// TwinCAT 3 PLC project UnitTests
// ProgramVersion: 3.1.4026.27
// libraries:
//   [ApplicationBase], * (Beckhoff Automation LLC)
//   Tc2_EtherCAT, * (Beckhoff Automation GmbH)
//   Tc2_Math, * (Beckhoff Automation GmbH)
//   Tc2_MC2, * (Beckhoff Automation GmbH)
//   Tc2_Standard, * (Beckhoff Automation GmbH)
//   Tc2_System, * (Beckhoff Automation GmbH)
//   Tc2_Utilities, * (Beckhoff Automation GmbH)
//   Tc3_EventLogger, * (Beckhoff Automation GmbH)
//   Tc3_PlcTestSuite, * (Simmel)
// project tree:
//   / TestsBase.TcPOU, TestsBaseTask.TcTTO
//   UnitTests/ADS/ ADS_TEST.TcPOU
//   UnitTests/Analog/ Analog_TEST.TcPOU
//   UnitTests/AnyBuffer/ AnyBuffer_TEST.TcPOU, GVL_TEST_AnyBuffer.TcGVL, TEST_AnyBuffer_Clear.TcPOU, TEST_AnyBuffer_DeleteAtIndex.TcPOU, TEST_AnyBuffer_InsertAtIndex.TcPOU, TEST_AnyBuffer_PeekAtIndex.TcPOU, TEST_AnyBuffer_PopAtIndex.TcPOU, TEST_AnyBuffer_PopLeft.TcPOU, TEST_AnyBuffer_PopRight.TcPOU, TEST_AnyBuffer_PushLeft.TcPOU, TEST_AnyBuffer_PushRight.TcPOU, TEST_AnyBuffer_ReplaceAtIndex.TcPOU
//   UnitTests/AnyBuffer/DUTs/ ST_TEST_AnyBuffer_Element.TcDUT
//   UnitTests/Axis/ Axis_Test.TcPOU
//   UnitTests/CollectionPeeker/ CollectionPeeker_Test.TcPOU
//   UnitTests/Collection/ Collection_TEST.TcPOU
//   UnitTests/ComponentCollection/ ComponentCollection_TEST.TcPOU
//   UnitTests/Component/ Component_TEST.TcPOU
//   UnitTests/CyclicComponent/ CyclicComponent_TEST.TcPOU
//   UnitTests/CyclicRunner/ CyclicRunner_TEST.TcPOU
//   UnitTests/Cylinder/ Cylinder_TEST.TcPOU
//   UnitTests/Digital/ DigitalInput_Combiner_TEST.TcPOU, DigitalInput_Debounce_TEST.TcPOU, DigitalInput_ForceVisitor_TEST.TcPOU, DigitalInput_NC_TEST.TcPOU, DigitalInput_NO_TEST.TcPOU, DigitalOutput_TEST.TcPOU
//   UnitTests/Events/ Events_TEST.TcPOU
//   UnitTests/EtherCat/ EtherCatMaster_TEST.TcPOU
//   UnitTests/Force/ ForcibleBool_TEST.TcPOU, ForcibleInt_Test.TcPOU
//   UnitTests/Initializer/ Initializer_TEST.TcPOU
//   UnitTests/List/ List_TEST.TcPOU
//   UnitTests/ModeChange/ ModeControl_TEST.TcPOU
//   UnitTests/ModuleCollection/ ModuleCollection_TEST.TcPOU
//   UnitTests/Module/ Module_TEST.TcPOU
//   UnitTests/Recipe/ Recipe_TEST.TcPOU, ST_Recipe.TcDUT
//   UnitTests/Safety/ SafetyBase_TEST.TcPOU
//   UnitTests/Serial/ SerialConnection_Tests.TcPOU
//   UnitTests/Statemachine/ Statemachine_TEST.TcPOU
//   UnitTests/Tracing/ Tracing_TEST.TcPOU
//   UnitTests/Utilities/ Utilities_TEST.TcPOU
//   _Mockups/AnyBuffer/ GVL_Samples_AnyBuffer.TcGVL, SampleFifo.TcPOU, SampleLifo.TcPOU, SampleList.TcPOU, SampleRing.TcPOU, Samples_AnyBuffer.TcPOU
//   _Mockups/CollectionPeeker/ CollectionPeeker_Mock.TcPOU
//   _Mockups/Collection/ Collection_Mockup.TcPOU, Item_Mockup.TcPOU
//   _Mockups/Components/ Component_Mockup.TcPOU, CyclicComponent_Mockup.TcPOU, InitializableComponent_Mockup.TcPOU, MockupComponentTcEvent.TcPOU
//   _Mockups/EtherCat/ EtherCatEventProvider_Mockup.TcPOU, EtherCatMaster_Mockup.TcPOU
//   _Mockups/ModeChange/ ModeControl_Mockup.TcPOU
//   _Mockups/Modules/ EquipmentModule_Mockup.TcPOU, MachineModule_Mockup.TcPOU, ModuleCollection_Mockup.TcPOU, Module_Mockup.TcPOU
//   _Mockups/SerialLineCtrl/ MockSerialLineCtrl.TcPOU
//   _Mockups/Statemachine/ StateMachineVisitor_Mockup.TcPOU, State_Mockup.TcPOU
//   _Mockups/Visitors/ ComponentVisitor_Mockup.TcPOU, GetSystemTreeNamesVisitor.TcPOU, ModuleVisitor_Mockup.TcPOU, QueryInterfaceResettables.TcPOU, StringCollection.TcPOU
// real-time tasks:
//   TASK UnitTestsBase: cycle T#10ms, priority 20, ADS port 350
//   TASK VFFS: cycle T#10ms, priority 21, ADS port 351
//   TASK PlcTask: cycle T#10ms, priority 22, ADS port 352
//   TASK Job Task: cycle default, priority 32
//   TASK MC-Task (MET): cycle T#2ms, priority 3, ADS port 521
//   TASK MC-Task (MPT): cycle T#10ms, priority 9, ADS port 531
// motion (NC):
//   TASK NC-Task 1 SAF: cycle T#2ms, priority 4, ADS port 501
//   TASK NC-Task 1 SVB: cycle T#10ms, priority 8, ADS port 511
//   AXIS TestAxis (id 1)
//     OtherSettings: AllowMotionCmdToSlave=true
//     encoder EncType=1
//     drive DrvType=5
//       Analog: TorqueSetpointScale=10, ScaleFactorActTorque=0.1
//     controller CtrType=1
//       CtrPara: PriorControlFactor=1
//         Observer: BandWidth=20
//   AXIS Unwind (id 2)
//     OtherSettings: AllowMotionCmdToSlave=true
//     encoder EncType=1
//     drive DrvType=5
//       Analog: TorqueSetpointScale=10, ScaleFactorActTorque=0.1
//       TimeComp: TaskDelayCycles=1
//     controller CtrType=1
//       CtrPara: PriorControlFactor=1
//         Observer: BandWidth=20
//   AXIS Seal (id 3)
//     OtherSettings: AllowMotionCmdToSlave=true
//     encoder EncType=1
//     drive DrvType=5
//       Analog: TorqueSetpointScale=10, ScaleFactorActTorque=0.1
//       TimeComp: TaskDelayCycles=1
//     controller CtrType=1
//       CtrPara: PriorControlFactor=1
//         Observer: BandWidth=20
//   AXIS Pull Wheel Left (id 4)
//     OtherSettings: AllowMotionCmdToSlave=true
//     encoder EncType=1
//     drive DrvType=5
//       Analog: TorqueSetpointScale=10, ScaleFactorActTorque=0.1
//       TimeComp: TaskDelayCycles=1
//     controller CtrType=1
//       CtrPara: PriorControlFactor=1
//         Observer: BandWidth=20
//   AXIS Pull Wheel Right (id 5)
//     OtherSettings: AllowMotionCmdToSlave=true
//     encoder EncType=1
//     drive DrvType=5
//       Analog: TorqueSetpointScale=10, ScaleFactorActTorque=0.1
//       TimeComp: TaskDelayCycles=1
//     controller CtrType=1
//       CtrPara: PriorControlFactor=1
//         Observer: BandWidth=20
// variable links:
//   (this object) <-> NC-Task 1 SAF/Axes/TestAxis
//     TestsBaseTask Inputs/TestsBase.Axis_Test.AxisRef.NcToPlc <-> Outputs/ToPlc
//     TestsBaseTask Outputs/TestsBase.Axis_Test.AxisRef.PlcToNc <-> Inputs/FromPlc
//   (this object) <-> UnitTests/UnitTests Instance
//     TestsBaseTask Inputs/TestsBase.SafetyBase_TEST.EStop_NOK.InfoData/Diag <-> TestsBaseTask Outputs/TestsBase.SafetyBase_TEST.InfoData_NOK/Diag
//     TestsBaseTask Inputs/TestsBase.SafetyBase_TEST.EStop_NOK.InfoData/State <-> TestsBaseTask Outputs/TestsBase.SafetyBase_TEST.InfoData_NOK/State
//     TestsBaseTask Inputs/TestsBase.SafetyBase_TEST.EStop_OK.InfoData/Diag <-> TestsBaseTask Outputs/TestsBase.SafetyBase_TEST.InfoData_OK/Diag
//     TestsBaseTask Inputs/TestsBase.SafetyBase_TEST.EStop_OK.InfoData/State <-> TestsBaseTask Outputs/TestsBase.SafetyBase_TEST.InfoData_OK/State
//     TestsBaseTask Inputs/TestsBase.SafetyBase_TEST.EStop_Sim.InfoData/Diag <-> TestsBaseTask Outputs/TestsBase.SafetyBase_TEST.InfoData_OK/Diag
//     TestsBaseTask Inputs/TestsBase.SafetyBase_TEST.EStop_Sim.InfoData/State <-> TestsBaseTask Outputs/TestsBase.SafetyBase_TEST.InfoData_OK/State
//     TestsBaseTask Inputs/TestsBase.SafetyBase_TEST.Group.InfoData/Diag <-> TestsBaseTask Outputs/TestsBase.SafetyBase_TEST.InfoData_Group/Diag
//     TestsBaseTask Inputs/TestsBase.SafetyBase_TEST.Group.InfoData/State <-> TestsBaseTask Outputs/TestsBase.SafetyBase_TEST.InfoData_Group/State
//     TestsBaseTask Inputs/TestsBase.SafetyBase_TEST.Reset <-> TestsBaseTask Outputs/TestsBase.SafetyBase_TEST.ResetPulse.Reset
//     TestsBaseTask Inputs/TestsBase.SafetyBase_TEST.Run <-> TestsBaseTask Outputs/TestsBase.SafetyBase_TEST.Group.Run
//     TestsBaseTask Outputs/TestsBase.SafetyBase_TEST.Group.Run <-> TestsBaseTask Inputs/TestsBase.SafetyBase_TEST.Run
//     TestsBaseTask Outputs/TestsBase.SafetyBase_TEST.InfoData_Group/Diag <-> TestsBaseTask Inputs/TestsBase.SafetyBase_TEST.Group.InfoData/Diag
//     TestsBaseTask Outputs/TestsBase.SafetyBase_TEST.InfoData_Group/State <-> TestsBaseTask Inputs/TestsBase.SafetyBase_TEST.Group.InfoData/State
//     TestsBaseTask Outputs/TestsBase.SafetyBase_TEST.InfoData_NOK/Diag <-> TestsBaseTask Inputs/TestsBase.SafetyBase_TEST.EStop_NOK.InfoData/Diag
//     TestsBaseTask Outputs/TestsBase.SafetyBase_TEST.InfoData_NOK/State <-> TestsBaseTask Inputs/TestsBase.SafetyBase_TEST.EStop_NOK.InfoData/State
//     TestsBaseTask Outputs/TestsBase.SafetyBase_TEST.InfoData_OK/Diag <-> TestsBaseTask Inputs/TestsBase.SafetyBase_TEST.EStop_OK.InfoData/Diag
//     TestsBaseTask Outputs/TestsBase.SafetyBase_TEST.InfoData_OK/Diag <-> TestsBaseTask Inputs/TestsBase.SafetyBase_TEST.EStop_Sim.InfoData/Diag
//     TestsBaseTask Outputs/TestsBase.SafetyBase_TEST.InfoData_OK/State <-> TestsBaseTask Inputs/TestsBase.SafetyBase_TEST.EStop_OK.InfoData/State
//     TestsBaseTask Outputs/TestsBase.SafetyBase_TEST.InfoData_OK/State <-> TestsBaseTask Inputs/TestsBase.SafetyBase_TEST.EStop_Sim.InfoData/State
//     TestsBaseTask Outputs/TestsBase.SafetyBase_TEST.ResetPulse.Reset <-> TestsBaseTask Inputs/TestsBase.SafetyBase_TEST.Reset
//   (this object) <-> MC Project1/Axes/Pull Wheel Left
//     PlcTask Inputs/MAIN.VFFS._PullWheels.PullWheelLeftAxisRef.McToPlc/Act <-> McToPlc/Act
//     PlcTask Inputs/MAIN.VFFS._PullWheels.PullWheelLeftAxisRef.McToPlc/Set <-> McToPlc/Set
//     PlcTask Inputs/MAIN.VFFS._PullWheels.PullWheelLeftAxisRef.McToPlc/Std <-> McToPlc/Std
//     PlcTask Outputs/MAIN.VFFS._PullWheels.PullWheelLeftAxisRef.PlcToMc/Std <-> PlcToMc/Std
//   (this object) <-> MC Project1/Axes/Pull Wheel Right
//     PlcTask Inputs/MAIN.VFFS._PullWheels.PullWheelRightAxisRef.McToPlc/Act <-> McToPlc/Act
//     PlcTask Inputs/MAIN.VFFS._PullWheels.PullWheelRightAxisRef.McToPlc/Set <-> McToPlc/Set
//     PlcTask Inputs/MAIN.VFFS._PullWheels.PullWheelRightAxisRef.McToPlc/Std <-> McToPlc/Std
//     PlcTask Outputs/MAIN.VFFS._PullWheels.PullWheelRightAxisRef.PlcToMc/Std <-> PlcToMc/Std
//   (this object) <-> MC Project1/Axes/Seal
//     PlcTask Inputs/MAIN.VFFS._Sealer.SealerAxisRef.McToPlc/Act <-> McToPlc/Act
//     PlcTask Inputs/MAIN.VFFS._Sealer.SealerAxisRef.McToPlc/Set <-> McToPlc/Set
//     PlcTask Inputs/MAIN.VFFS._Sealer.SealerAxisRef.McToPlc/Std <-> McToPlc/Std
//     PlcTask Outputs/MAIN.VFFS._Sealer.SealerAxisRef.PlcToMc/Std <-> PlcToMc/Std
//   (this object) <-> MC Project1/Axes/Unwind
//     PlcTask Inputs/MAIN.VFFS._Unwind.UnwindAxisRef.McToPlc/Act <-> McToPlc/Act
//     PlcTask Inputs/MAIN.VFFS._Unwind.UnwindAxisRef.McToPlc/Set <-> McToPlc/Set
//     PlcTask Inputs/MAIN.VFFS._Unwind.UnwindAxisRef.McToPlc/Std <-> McToPlc/Std
//     PlcTask Outputs/MAIN.VFFS._Unwind.UnwindAxisRef.PlcToMc/Std <-> PlcToMc/Std

CONFIGURATION UnitTests
    RESOURCE PLC ON TwinCAT3
        TASK TestsBaseTask(INTERVAL := T#10ms, PRIORITY := 20);
        PROGRAM TestsBase WITH TestsBaseTask : TestsBase;
    END_RESOURCE
END_CONFIGURATION

// ---- UnitTests/AnyBuffer/DUTs/ST_TEST_AnyBuffer_Element.TcDUT
TYPE ST_TEST_AnyBuffer_Element :
STRUCT
	id				: INT;
	name			: STRING;
END_STRUCT
END_TYPE

// ---- UnitTests/Recipe/ST_Recipe.TcDUT
TYPE ST_Recipe :
	STRUCT
		ValueA : LREAL;
		ValueB : DINT;
		ValueC : BOOL;
	END_STRUCT
END_TYPE

// ---- UnitTests/AnyBuffer/GVL_TEST_AnyBuffer.TcGVL
VAR_GLOBAL
	// System Under Test (SUT)
    RawBuffer       		: ARRAY[TEST_LL..TEST_UL] OF DINT;
    fbAnyBuffer    			: AnyBuffer(pBuffer := RawBuffer,
									bufferBoundLower := TEST_LL,
									bufferBoundUpper := TEST_UL,
									isBufferPersistent := FALSE);

	// Compare buffer
	CompareBuffer : ARRAY[TEST_LL..TEST_UL] OF DINT;
	fbCompareBuffer : AnyBuffer(pBuffer := CompareBuffer,
								bufferBoundLower := TEST_LL,
								bufferBoundUpper := TEST_UL,
								isBufferPersistent := FALSE);

    // Test Variables
    Success         		: BOOL;
	AppendedElement			: DINT;
	ReturnedElement			: DINT;
	WrongSizeElement		: INT;
	testElement				: DINT;

	// Bool
	TEST_BOOL_TRUE			: BOOL := TRUE;
	TEST_BOOL_FALSE			: BOOL := FALSE;
	TEST_DINT				: DINT;
	TEST_REAL				: REAL;
END_VAR
VAR_GLOBAL CONSTANT
	// Changing the limits is allowed, but the tests are built for an array size 5 elements
	TEST_LL					: INT := 0;
	TEST_UL					: INT := 4;
END_VAR

// ---- _Mockups/AnyBuffer/GVL_Samples_AnyBuffer.TcGVL
VAR_GLOBAL PERSISTENT
	buffer					: ARRAY[S_LL..S_UL] OF ST_TEST_AnyBuffer_Element;			// Any size buffer of any type
END_VAR

VAR_GLOBAL
	anyBuffer				: AnyBuffer(buffer, S_LL, S_UL, TRUE); 		// persistent buffer handler
END_VAR

VAR_GLOBAL CONSTANT
	S_LL					: INT := 0;
	S_UL					: INT := 2;
END_VAR

// ---- TestsBase.TcPOU
PROGRAM TestsBase
VAR
	CyclicRunner_TEST			   : CyclicRunner_TEST;
	ComponentCollection_TEST	   : ComponentCollection_TEST;
	Module_TEST					   : Module_TEST;
	CyclicComponent_TEST		   : CyclicComponent_TEST;
	Component_TEST				   : Component_TEST;
	ModuleCollection_TEST		   : ModuleCollection_TEST;
	Tracing_TEST				   : Tracing_TEST;
	Initializer_TEST			   : Initializer_TEST;
	Events_TEST					   : Events_TEST;
	Statemachine_TEST			   : Statemachine_TEST;
	Collection_Test				   : Collection_TEST();
	List_TEST					   : List_TEST;
	ModeControl_TEST			   : ModeControl_TEST;
	CollectionPeeker_Test		   : CollectionPeeker_Test;
	ForcibleBool_TEST			   : ForcibleBool_TEST;
	ForcibleInt_Test			   : ForcibleInt_Test;
	Utilities_TEST				   : Utilities_TEST;
	DigitalInput_NC_TEST		   : DigitalInput_NC_TEST;
	DigitalInput_NO_TEST		   : DigitalInput_NO_TEST;
	DigitalOutput_TEST			   : DigitalOutput_TEST;
	DigitalInput_Combiner_TEST	   : DigitalInput_Combiner_TEST;
	DigitalInput_Debounce_TEST	   : DigitalInput_Debounce_TEST;
	Cylinder_TEST				   : Cylinder_TEST;
	SafetyBase_TEST				   : SafetyBase_TEST;
	ADS_TEST					   : ADS_TEST;
	DigitalInput_ForceVisitor_TEST : DigitalInput_ForceVisitor_TEST;
	Recipe_TEST					   : Recipe_TEST;
	Analog_TEST					   : Analog_TEST;
	Serial_TEST					   : SerialConnection_Tests;
	Axis_Test					   : Axis_Test;
	EtherCatMaster_TEST		   : EtherCatMaster_TEST;

	//
	Component1				  : CyclicComponent_Mockup('Component 1');
	Component2				  : CyclicComponent_Mockup('Component 2');
	Component3				  : CyclicComponent_Mockup('Component 3');
	Component4				  : CyclicComponent_Mockup('Component 4');
	Em						  : EquipmentModule_Mockup('Em', Component1, Component2);
	EmEm					  : MachineModule_Mockup('EmEm', Em, Component3, Component4);
	EmEmEm					  : MachineModule_Mockup('EmEmEm', EmEm, Component3, Component4);
	Machine					  : MachineModule_Mockup('Machine', EmEmEm, Component3, Component4);
	StringCollection		  : StringCollection<100>;
	MachineModuleVisitor	  : GetSystemTreeNamesVisitor(StringCollection);
	QueryInterfaceResettables : QueryInterfaceResettables();
	Rerun					  : BOOL;
END_VAR

GlobalTestSuite.TestSuite.TestSuiteName := 'Application Base Test Suite';
Tracing_TEST();
CyclicRunner_TEST();
ComponentCollection_TEST();
Module_TEST();
Component_TEST();
CyclicComponent_TEST();
ModuleCollection_TEST();
Initializer_TEST();
Events_TEST();
Statemachine_TEST();
Collection_Test();
List_TEST();
ModeControl_TEST();
CollectionPeeker_Test();
ForcibleBool_TEST();
Utilities_TEST();
DigitalInput_NC_TEST();
DigitalInput_NO_TEST();
DigitalOutput_TEST();
DigitalInput_Combiner_TEST();
DigitalInput_Debounce_TEST();
Cylinder_TEST();
SafetyBase_TEST();
ADS_TEST();
DigitalInput_ForceVisitor_TEST();
Recipe_TEST();
Analog_TEST();
AnyBuffer_TEST();
ForcibleInt_Test();
Serial_TEST();
Axis_Test();
EtherCatMaster_TEST();

// Mockup code
Samples_AnyBuffer();
//
IF NOT Machine.Initialized THEN
	Machine.Initialize();
ELSE
	Machine.CyclicLogic();
	MachineModuleVisitor.GetTree(Machine);
	QueryInterfaceResettables.GetAllResetComponents(Em);
END_IF

IF Rerun THEN
	Rerun := FALSE;
	GlobalTestSuite.TestSuite.ReRunTests();
END_IF

END_PROGRAM

// ---- UnitTests/CyclicRunner/CyclicRunner_TEST.TcPOU
FUNCTION_BLOCK CyclicRunner_TEST
VAR
END_VAR

AddTwoCyclicCalleesAndRun();
CollectionAddsCyclicSucessfully();
CollectionRejectsAddingCyclicDuplicate();
CollectionRejectsAddingNullCyclic();
CollectionRejectsAddingTooManyCyclics();
CollectionRejectsRemoveWhenEmpty();
CollectionRejectsRemoveWhenNotFound();
CollectionRejectsRemovingNullCyclic();
CollectionRemovesCyclicSuccessfully();

METHOD AddTwoCyclicCalleesAndRun
VAR
	Expected	 : BOOL := TRUE;
	Actual		 : BOOL;
	CyclicRunner : CyclicRunner<ApplicationBaseParameter.MaxCountInCollections>;
	Component	 : ARRAY[0..1] OF CyclicComponent_Mockup[(Name := 'Component 1'), (Name := 'Component 2')];
END_VAR
IF TestSuite.Test(__POUNAME()).ExecuteTest() THEN
	CyclicRunner.AddCallee(Component[0]);
	CyclicRunner.AddCallee(Component[1]);
	CyclicRunner.CallAll();
	Actual := Component[0].WasCalled AND Component[1].WasCalled;
	TestSuite.Test(__POUNAME()).AssertEqual(Expected, Actual);
END_IF
END_METHOD

METHOD CollectionAddsCyclicSucessfully
VAR
	Expected	   : BOOL := TRUE;
	Actual		   : BOOL;
	CyclicRunner : CyclicRunner<ApplicationBaseParameter.MaxCountInCollections>;
	Cyclic	 : CyclicComponent_Mockup(Name := 'Cyclic 1');
END_VAR
IF TestSuite.Test(__POUNAME()).ExecuteTest() THEN
	Actual := CyclicRunner.AddCallee(Cyclic) = RegistrationResult.Succeeded;
	TestSuite.Test(__POUNAME()).AssertEqual(Expected, Actual);
END_IF
END_METHOD

METHOD CollectionRejectsAddingCyclicDuplicate
VAR
	Expected	   : BOOL := TRUE;
	Actual		   : BOOL;
	CyclicRunner : CyclicRunner<ApplicationBaseParameter.MaxCountInCollections>;
	Cyclic	 : CyclicComponent_Mockup(Name := 'Cyclic 1');
END_VAR
IF TestSuite.Test(__POUNAME()).ExecuteTest() THEN
	CyclicRunner.AddCallee(Cyclic);
	Actual := CyclicRunner.AddCallee(Cyclic) = RegistrationResult.AlreadyAdded;
	TestSuite.Test(__POUNAME()).AssertEqual(Expected, Actual);
END_IF
END_METHOD

METHOD CollectionRejectsAddingNullCyclic
VAR
	Expected	   : BOOL := TRUE;
	Actual		   : BOOL;
	CyclicRunner : CyclicRunner<ApplicationBaseParameter.MaxCountInCollections>;
END_VAR
IF TestSuite.Test(__POUNAME()).ExecuteTest() THEN
	Actual := CyclicRunner.AddCallee(16#0) = RegistrationResult.NullReference;
	TestSuite.Test(__POUNAME()).AssertEqual(Expected, Actual);
END_IF
END_METHOD

METHOD CollectionRejectsAddingTooManyCyclics
VAR
	Expected	   : BOOL := TRUE;
	Actual		   : BOOL;
	CyclicRunner : CyclicRunner<1>;
	Cyclic1	 : CyclicComponent_Mockup(Name := 'Cyclic 1');
	Cyclic2	 : CyclicComponent_Mockup(Name := 'Cyclic 2');
END_VAR
IF TestSuite.Test(__POUNAME()).ExecuteTest() THEN
	CyclicRunner.AddCallee(Cyclic1);
	Actual := CyclicRunner.AddCallee(Cyclic2) = RegistrationResult.TooManyComponents;
	TestSuite.Test(__POUNAME()).AssertEqual(Expected, Actual);
END_IF
END_METHOD

METHOD CollectionRejectsRemoveWhenEmpty
VAR
	Expected	   : BOOL := TRUE;
	Actual		   : BOOL;
	CyclicRunner : CyclicRunner<ApplicationBaseParameter.MaxCountInCollections>;
	Cyclic1	 : CyclicComponent_Mockup(Name := 'Cyclic 1');
END_VAR
IF TestSuite.Test(__POUNAME()).ExecuteTest() THEN
	Actual := CyclicRunner.RemoveCallee(Cyclic1) = RegistrationResult.CollectionEmpty;
	TestSuite.Test(__POUNAME()).AssertEqual(Expected, Actual);
END_IF
END_METHOD

METHOD CollectionRejectsRemoveWhenNotFound
VAR
	Expected	   : BOOL := TRUE;
	Actual		   : BOOL;
	CyclicRunner : CyclicRunner<ApplicationBaseParameter.MaxCountInCollections>;
	Cyclic1	 : CyclicComponent_Mockup(Name := 'Cyclic 1');
	Cyclic2	 : CyclicComponent_Mockup(Name := 'Cyclic 2');
END_VAR
IF TestSuite.Test(__POUNAME()).ExecuteTest() THEN
	CyclicRunner.AddCallee(Cyclic1);
	Actual := CyclicRunner.RemoveCallee(Cyclic2) = RegistrationResult.NotFoundInCollection;
	TestSuite.Test(__POUNAME()).AssertEqual(Expected, Actual);
END_IF
END_METHOD

METHOD CollectionRejectsRemovingNullCyclic
VAR
	Expected	   : BOOL := TRUE;
	Actual		   : BOOL;
	CyclicRunner : CyclicRunner<ApplicationBaseParameter.MaxCountInCollections>;
END_VAR
IF TestSuite.Test(__POUNAME()).ExecuteTest() THEN
	Actual := CyclicRunner.RemoveCallee(16#0) = RegistrationResult.NullReference;
	TestSuite.Test(__POUNAME()).AssertEqual(Expected, Actual);
END_IF
END_METHOD

METHOD CollectionRemovesCyclicSuccessfully
VAR
	Expected	   : BOOL := TRUE;
	Actual		   : BOOL;
	CyclicCollection : CyclicRunner<ApplicationBaseParameter.MaxCountInCollections>;
	Cyclic		: CyclicComponent_Mockup(Name := 'Component 1');
	AddedCyclic : I_Cyclic := Cyclic;
	CollectionCyclic : I_Cyclic;
END_VAR
IF TestSuite.Test(__POUNAME()).ExecuteTest() THEN
	CyclicCollection.AddCallee(Cyclic);
	Actual := CyclicCollection.RemoveCallee(Cyclic) = RegistrationResult.Succeeded;
	TestSuite.Test(__POUNAME()).AssertEqual(Expected, Actual);
END_IF
END_METHOD

END_FUNCTION_BLOCK

// ---- _Mockups/Components/CyclicComponent_Mockup.TcPOU
FUNCTION_BLOCK CyclicComponent_Mockup EXTENDS CyclicComponent IMPLEMENTS I_Resettable
VAR
	_WasCalled : BOOL;
END_VAR

METHOD CyclicLogic
_WasCalled := TRUE;
END_METHOD

METHOD Reset
END_METHOD

PROPERTY WasCalled : BOOL
GET
WasCalled := _WasCalled;
END_GET
END_PROPERTY

END_FUNCTION_BLOCK

// ---- UnitTests/ComponentCollection/ComponentCollection_TEST.TcPOU
FUNCTION_BLOCK ComponentCollection_TEST
VAR

END_VAR

CollectionAddsComponentSucessfully();
CollectionRejectsAddingComponentDuplicate();
CollectionRejectsAddingNullComponent();
CollectionRejectsAddingTooManyComponents();
CollectionRejectsRemoveWhenEmpty();
CollectionRejectsRemoveWhenNotFound();
CollectionRejectsRemovingNullComponent();
CollectionReturnsComponentByName();
CollectionRemovesComponentSuccessfully();
CollectionGetItemAtIndex();
CollectionGetCount();

METHOD CollectionAddsComponentSucessfully
VAR
	Expected			: BOOL := TRUE;
	Actual				: BOOL;
	ComponentCollection : ComponentCollection<ApplicationBaseParameter.MaxCountInCollections>;
	Component			: CyclicComponent_Mockup(Name := 'Component 1');
END_VAR
IF TestSuite.Test(__POUNAME()).ExecuteTest() THEN
	Actual := ComponentCollection.AddComponent(Component) = RegistrationResult.Succeeded;
	TestSuite.Test(__POUNAME()).AssertEqual(Expected, Actual);
END_IF
END_METHOD

METHOD CollectionGetCount
VAR
	Expected			: UDINT;
	Actual				: UDINT;
	ComponentCollection : ComponentCollection<ApplicationBaseParameter.MaxCountInCollections>;
	Component			: CyclicComponent_Mockup(Name := 'Component 1');
END_VAR
IF TestSuite.Test(__POUNAME()).ExecuteTest() THEN
	Expected := 1;
	ComponentCollection.AddComponent(Component);
	Actual := ComponentCollection.Count;
	TestSuite.Test(__POUNAME()).AssertEqual(Expected, Actual);
END_IF
END_METHOD

METHOD CollectionGetItemAtIndex
VAR
	Expected			: BOOL := TRUE;
	Actual				: BOOL;
	ComponentCollection : ComponentCollection<2>;
	Component1			: CyclicComponent_Mockup(Name := 'Component 1');
	Component2			: CyclicComponent_Mockup(Name := 'Component 2');
	ReturnedComponent	: I_Component;
END_VAR
IF TestSuite.Test(__POUNAME()).ExecuteTest() THEN
	ComponentCollection.AddComponent(Component1);
	ComponentCollection.AddComponent(Component2);
	ReturnedComponent := ComponentCollection.GetAtIndex(1);
	Actual			  := ReturnedComponent.Name = Component2.Name;
	TestSuite.Test(__POUNAME()).AssertEqual(Expected, Actual);
END_IF
END_METHOD

METHOD CollectionRejectsAddingComponentDuplicate
VAR
	Expected	   : BOOL := TRUE;
	Actual		   : BOOL;
	ComponentCollection : ComponentCollection<ApplicationBaseParameter.MaxCountInCollections>;
	Component			: CyclicComponent_Mockup(Name := 'Component 1');
END_VAR
IF TestSuite.Test(__POUNAME()).ExecuteTest() THEN
	ComponentCollection.AddComponent(Component);
	Actual := ComponentCollection.AddComponent(Component) = RegistrationResult.AlreadyAdded;
	TestSuite.Test(__POUNAME()).AssertEqual(Expected, Actual);
END_IF
END_METHOD

METHOD CollectionRejectsAddingNullComponent
VAR
	Expected	   : BOOL := TRUE;
	Actual		   : BOOL;
	ComponentCollection : ComponentCollection<ApplicationBaseParameter.MaxCountInCollections>;
END_VAR
IF TestSuite.Test(__POUNAME()).ExecuteTest() THEN
	Actual := ComponentCollection.AddComponent(16#0) = RegistrationResult.NullReference;
	TestSuite.Test(__POUNAME()).AssertEqual(Expected, Actual);
END_IF
END_METHOD

METHOD CollectionRejectsAddingTooManyComponents
VAR
	Expected	   : BOOL := TRUE;
	Actual		   : BOOL;
	ComponentCollection : ComponentCollection<1>;
	Component1			: CyclicComponent_Mockup(Name := 'Component 1');
	Component2			: CyclicComponent_Mockup(Name := 'Component 2');
END_VAR
IF TestSuite.Test(__POUNAME()).ExecuteTest() THEN
	ComponentCollection.AddComponent(Component1);
	Actual := ComponentCollection.AddComponent(Component2) = RegistrationResult.TooManyComponents;
	TestSuite.Test(__POUNAME()).AssertEqual(Expected, Actual);
END_IF
END_METHOD

METHOD CollectionRejectsRemoveWhenEmpty
VAR
	Expected	   : BOOL := TRUE;
	Actual		   : BOOL;
	ComponentCollection : ComponentCollection<ApplicationBaseParameter.MaxCountInCollections>;
	Component			: CyclicComponent_Mockup(Name := 'Component 1');
END_VAR
IF TestSuite.Test(__POUNAME()).ExecuteTest() THEN
	Actual := ComponentCollection.RemoveComponent(Component) = RegistrationResult.CollectionEmpty;
	TestSuite.Test(__POUNAME()).AssertEqual(Expected, Actual);
END_IF
END_METHOD

METHOD CollectionRejectsRemoveWhenNotFound
VAR
	Expected	   : BOOL := TRUE;
	Actual		   : BOOL;
	ComponentCollection : ComponentCollection<1>;
	Component1			: CyclicComponent_Mockup(Name := 'Component 1');
	Component2			: CyclicComponent_Mockup(Name := 'Component 2');
END_VAR
IF TestSuite.Test(__POUNAME()).ExecuteTest() THEN
	ComponentCollection.AddComponent(Component1);
	Actual := ComponentCollection.RemoveComponent(Component2) = RegistrationResult.NotFoundInCollection;
	TestSuite.Test(__POUNAME()).AssertEqual(Expected, Actual);
END_IF
END_METHOD

METHOD CollectionRejectsRemovingNullComponent
VAR
	Expected	   : BOOL := TRUE;
	Actual		   : BOOL;
	ComponentCollection : ComponentCollection<ApplicationBaseParameter.MaxCountInCollections>;
END_VAR
IF TestSuite.Test(__POUNAME()).ExecuteTest() THEN
	Actual := ComponentCollection.RemoveComponent(16#0) = RegistrationResult.NullReference;
	TestSuite.Test(__POUNAME()).AssertEqual(Expected, Actual);
END_IF
END_METHOD

METHOD CollectionRemovesComponentSuccessfully
VAR
	Expected			: BOOL := TRUE;
	Actual				: BOOL;
	ComponentCollection : ComponentCollection<ApplicationBaseParameter.MaxCountInCollections>;
	Component			: CyclicComponent_Mockup(Name := 'Component 1');
	AddedComponent		: I_Component := Component;
	CollectionComponent : I_Component;
END_VAR
IF TestSuite.Test(__POUNAME()).ExecuteTest() THEN
	ComponentCollection.AddComponent(Component);
	CollectionComponent := ComponentCollection.GetComponentByName('Component 1');
	IF CollectionComponent = AddedComponent THEN
		Actual := ComponentCollection.RemoveComponent(Component) = RegistrationResult.Succeeded;
	END_IF
	TestSuite.Test(__POUNAME()).AssertEqual(Expected, Actual);
END_IF
END_METHOD

METHOD CollectionReturnsComponentByName
VAR
	Expected	   : STRING := 'Component 1';
	Actual		   : STRING;
	ComponentCollection : ComponentCollection<ApplicationBaseParameter.MaxCountInCollections>;
	Component			: CyclicComponent_Mockup(Name := 'Component 1');
END_VAR
IF TestSuite.Test(__POUNAME()).ExecuteTest() THEN
	ComponentCollection.AddComponent(Component);
	Actual := ComponentCollection.GetComponentByName(Expected).Name;
	TestSuite.Test(__POUNAME()).AssertEqual(Expected, Actual);
END_IF
END_METHOD

END_FUNCTION_BLOCK

// ---- UnitTests/Module/Module_TEST.TcPOU
FUNCTION_BLOCK Module_TEST
VAR
	
END_VAR

OnCyclicCallCalled();
RegisterComponentRegistered();
RegisterCyclicRegistered();
RegisterModuleRegistered();
RegisterWithParentRegistered();
CheckVisitComponentsMechanismAndGetVisitedCount();
CheckVisitModulesMechanismAndGetVisitedCount();
RegisterInitializeRegistered();
CallInitializationMethod();
NameAssigned();
DeregisterWithParent();

METHOD CallInitializationMethod
VAR_INST
	Expected			   : BOOL;
	Actual				   : BOOL;
END_VAR
VAR
	InitializableComponent : InitializableComponent_Mockup('Component 1');
	Module				   : Module_Mockup('Module');
END_VAR
IF TestSuite.Test(__POUNAME()).ExecuteTest() THEN
	Expected						   := TRUE;
	InitializableComponent.Initialized := TRUE;
	Module.RegisterInitialize(InitializableComponent);
	Module.Initialize();
	Actual := Module.Initialized;
	TestSuite.Test(__POUNAME()).AssertEqual(Expected, Actual);
END_IF
END_METHOD

METHOD CheckVisitComponentsMechanismAndGetVisitedCount
VAR_INST
	Expected : DINT;
	Actual	 : DINT;
END_VAR
VAR
	Component1		 : CyclicComponent_Mockup('Component 1');
	Component2		 : CyclicComponent_Mockup('Component 2');
	Module			 : EquipmentModule_Mockup('Module 1', Component1, Component2);
	StringCollection : StringCollection<100>;
	ComponentVisitor : ComponentVisitor_Mockup(StringCollection);
END_VAR
IF TestSuite.Test(__POUNAME()).ExecuteTest() THEN
	Expected := 2;
	Module.CyclicLogic();
	Module.Components.Accept(ComponentVisitor);
	Actual := StringCollection.Entries;
	TestSuite.Test(__POUNAME()).AssertEqual(Expected, Actual);
END_IF
END_METHOD

METHOD CheckVisitModulesMechanismAndGetVisitedCount
VAR_INST
	Expected : DINT;
	Actual	 : DINT;
END_VAR
VAR
	Component1		 : CyclicComponent_Mockup('Component 1');
	Component2		 : CyclicComponent_Mockup('Component 2');
	Module			 : EquipmentModule_Mockup('Module 1', Component1, Component2);
	StringCollection : StringCollection<100>;
	ComponentVisitor : ComponentVisitor_Mockup(StringCollection);

	//
	Component3	  : CyclicComponent_Mockup('Component 3');
	Component4	  : CyclicComponent_Mockup('Component 4');
	ModuleEm	  : EquipmentModule_Mockup('Module', Component1, Component2);
	Machine		  : MachineModule_Mockup('Machine', ModuleEm, Component3, Component4);
	ModuleVisitor : ModuleVisitor_Mockup(StringCollection);
END_VAR
IF TestSuite.Test(__POUNAME()).ExecuteTest() THEN
	Expected := 1;
	StringCollection.Clear();
	Machine.CyclicLogic();
	Machine.Modules.Accept(ModuleVisitor);
	Actual := StringCollection.Entries;
	TestSuite.Test(__POUNAME()).AssertEqual(Expected, Actual);
END_IF
END_METHOD

METHOD DeregisterWithParent
VAR_INST
	Expected	   : BOOL;
	Actual		   : BOOL;
	ExpectedModule : I_Module;
	ActualModule   : I_Module;
END_VAR
VAR
	Component1		 : CyclicComponent_Mockup('Component 1');
	Component2		 : CyclicComponent_Mockup('Component 2');
	StringCollection : StringCollection<100>;
	Component3	  : CyclicComponent_Mockup('Component 3');
	Component4	  : CyclicComponent_Mockup('Component 4');
	ModuleEm	  : EquipmentModule_Mockup('Module', Component1, Component2);
	Machine		  : MachineModule_Mockup('Machine', ModuleEm, Component3, Component4);
END_VAR
IF TestSuite.Test(__POUNAME()).ExecuteTest() THEN
	Expected	   := TRUE;
	ExpectedModule := 0;
	ModuleEm.DeregisterWithParent(Machine);
	ActualModule := Machine.GetModuleByName('Module');
	Actual		 := ExpectedModule = ActualModule;
	TestSuite.Test(__POUNAME()).AssertEqual(Expected, Actual);
END_IF
END_METHOD

METHOD NameAssigned
VAR_INST
	Expected : STRING;
	Actual	 : STRING;
	//Module	 : Module_Mockup('Module');
END_VAR
VAR
	Component1		 : CyclicComponent_Mockup('Component 1');
	Component2		 : CyclicComponent_Mockup('Component 2');
	Module			 : EquipmentModule_Mockup('Module 1', Component1, Component2);
END_VAR
IF TestSuite.Test(__POUNAME()).ExecuteTest() THEN
	Expected := 'Module 1';
	Actual	 := Module.Name;
	TestSuite.Test(__POUNAME()).AssertEqual(Expected, Actual);
END_IF
END_METHOD

METHOD OnCyclicCallCalled
VAR_INST
	Expected		: BOOL;
	Actual			: BOOL;
END_VAR
VAR
	CyclicComponent : CyclicComponent_Mockup('Component 1');
	Module			: Module_Mockup('Module');
END_VAR
IF TestSuite.Test(__POUNAME()).ExecuteTest() THEN
	Expected := TRUE;
	Module.RegisterCyclic(CyclicComponent);
	Module.CyclicLogic();
	Actual := CyclicComponent.WasCalled;
	TestSuite.Test(__POUNAME()).AssertEqual(Expected, Actual);
END_IF
END_METHOD

METHOD RegisterComponentRegistered
VAR_INST
	Expected		: BOOL;
	Actual			: BOOL;
END_VAR
VAR
	CyclicComponent : CyclicComponent_Mockup('Component 1');
	Module			: Module_Mockup('Module');
	BaseComponent	: I_Component;
	AddedComponent	: I_Component;
END_VAR
IF TestSuite.Test(__POUNAME()).ExecuteTest() THEN
	Expected	  := TRUE;
	BaseComponent := CyclicComponent;
	Module.RegisterComponent(CyclicComponent);
	Module.CyclicLogic();
	AddedComponent := Module.GetComponentByName('Component 1');
	Actual		   := BaseComponent = AddedComponent;
	TestSuite.Test(__POUNAME()).AssertEqual(Expected, Actual);
END_IF
END_METHOD

METHOD RegisterCyclicRegistered
VAR_INST
	Expected		: BOOL;
	Actual			: BOOL;
END_VAR
VAR
	CyclicComponent : CyclicComponent_Mockup('Component 1');
	Module			: Module_Mockup('Module');
END_VAR
IF TestSuite.Test(__POUNAME()).ExecuteTest() THEN
	Expected := TRUE;
	Module.RegisterCyclic(CyclicComponent);
	Module.CyclicLogic();
	Actual := CyclicComponent.WasCalled;
	TestSuite.Test(__POUNAME()).AssertEqual(Expected, Actual);
END_IF
END_METHOD

METHOD RegisterInitializeRegistered
VAR_INST
	Expected			   : BOOL;
	Actual				   : BOOL;
END_VAR
VAR
	InitializableComponent : InitializableComponent_Mockup('Component 1');
	Module				   : Module_Mockup('Module');
END_VAR
IF TestSuite.Test(__POUNAME()).ExecuteTest() THEN
	Expected		   := TRUE;
	Module.Initialized := TRUE;
	Module.RegisterInitialize(InitializableComponent);
	Module.Initialize();
	Actual := InitializableComponent.InitializeWasCalled;
	TestSuite.Test(__POUNAME()).AssertEqual(Expected, Actual);
END_IF
END_METHOD

METHOD RegisterModuleRegistered
VAR_INST
	Expected		 : BOOL;
	Actual			 : BOOL;
END_VAR
VAR
	BaseModule		 : I_Module;
	AddedModule		 : I_Module;
	EquipmentModule	 : Module_Mockup('EquipmentModule');
	EquipmentModule2 : Module_Mockup('EquipmentModule2');
END_VAR
IF TestSuite.Test(__POUNAME()).ExecuteTest() THEN
	Expected   := TRUE;
	BaseModule := EquipmentModule;
	EquipmentModule2.RegisterModule(EquipmentModule);
	AddedModule := EquipmentModule2.GetModuleByName('EquipmentModule');
	Actual		:= BaseModule = AddedModule;
	TestSuite.Test(__POUNAME()).AssertEqual(Expected, Actual);
END_IF
END_METHOD

METHOD RegisterWithParentRegistered
VAR_INST
	Expected	   : BOOL;
	Actual		   : BOOL;
	ExpectedModule : I_Module;
	ActualModule   : I_Module;
END_VAR
VAR
	Component1		 : CyclicComponent_Mockup('Component 1');
	Component2		 : CyclicComponent_Mockup('Component 2');
	Component3	  : CyclicComponent_Mockup('Component 3');
	Component4	  : CyclicComponent_Mockup('Component 4');
	ModuleEm	  : EquipmentModule_Mockup('Module', Component1, Component2);
	Machine		  : MachineModule_Mockup('Machine', ModuleEm, Component3, Component4);
END_VAR
IF TestSuite.Test(__POUNAME()).ExecuteTest() THEN
	Expected	   := TRUE;
	ExpectedModule := ModuleEm;
	Machine.CyclicLogic();
	ActualModule := Machine.GetModuleByName('Module');
	Actual		 := ExpectedModule = ActualModule;
	TestSuite.Test(__POUNAME()).AssertEqual(Expected, Actual);
END_IF
END_METHOD

END_FUNCTION_BLOCK

// ---- _Mockups/Components/InitializableComponent_Mockup.TcPOU
FUNCTION_BLOCK InitializableComponent_Mockup EXTENDS CyclicComponent IMPLEMENTS I_Initializable
VAR
	_Initialized		 : BOOL;
	_WasCalled			 : BOOL;
	_InitializeWasCalled : BOOL;
END_VAR

METHOD CyclicLogic
_WasCalled := TRUE;
END_METHOD

METHOD Initialize
_InitializeWasCalled := TRUE;
END_METHOD

{attribute 'monitoring' := 'call'}
PROPERTY Initialized : BOOL
GET
Initialized := _Initialized;
END_GET
SET
_Initialized := Initialized;
END_SET
END_PROPERTY

PROPERTY InitializeWasCalled : BOOL
GET
InitializeWasCalled := _InitializeWasCalled;
END_GET
END_PROPERTY

PROPERTY WasCalled : BOOL
GET
WasCalled := _WasCalled;
END_GET
END_PROPERTY

END_FUNCTION_BLOCK

// ---- _Mockups/Modules/Module_Mockup.TcPOU
FUNCTION_BLOCK Module_Mockup EXTENDS Module
VAR
	_WasCalled : BOOL;
END_VAR

METHOD GetComponentByName : I_Component
VAR_INPUT
	Name : T_MaxString;
END_VAR
GetComponentByName := ComponentCollection.GetComponentByName(Name);
END_METHOD

METHOD GetModuleByName : I_Module
VAR_INPUT
	Module : T_MaxString;
END_VAR
GetModuleByName := ModuleCollection.GetModuleByName(Module);
END_METHOD

(* This Module will be done initializeing when ModuleInitialized := TRUE;, subequently all subitems will be called to be initialized*)
METHOD Initializing
ModuleInitialized := TRUE;
END_METHOD

METHOD OnCyclicCall
END_METHOD

PROPERTY WasCalled : BOOL
GET
WasCalled := _WasCalled;
END_GET
END_PROPERTY

END_FUNCTION_BLOCK

// ---- _Mockups/Modules/EquipmentModule_Mockup.TcPOU
FUNCTION_BLOCK EquipmentModule_Mockup EXTENDS Module
VAR
	SubModule	   : I_Module;
	TestComponent1 : I_Component;
	TestComponent2 : I_Component;
END_VAR

//FB_Init is always available implicitly and it is used primarily for initialization.

//The return value is not evaluated. For a specific influence, you can also declare the

//methods explicitly and provide additional code there with the standard initialization

//code. You can evaluate the return value.
METHOD FB_Init : BOOL
VAR_INPUT
	bInitRetains   : BOOL; // TRUE: the retain variables are initialized (reset warm / reset cold)
	bInCopyCode	   : BOOL; // TRUE: the instance will be copied to the copy code afterward (online change)   
	Name		   : T_MaxString;
	TestComponent1 : I_Component;
	TestComponent2 : I_Component;
END_VAR
THIS^.TestComponent1 := TestComponent1;
THIS^.TestComponent2 := TestComponent2;
TestComponent1.RegisterWithParent(THIS^);
TestComponent2.RegisterWithParent(THIS^);
END_METHOD

METHOD GetComponentByName : I_Component
VAR_INPUT
	Name : T_MaxString;
END_VAR
GetComponentByName := ComponentCollection.GetComponentByName(Name);
END_METHOD

METHOD GetModuleByName : I_Module
VAR_INPUT
	Module : T_MaxString;
END_VAR
GetModuleByName := ModuleCollection.GetModuleByName(Module);
END_METHOD

(* This Module will be done initializeing when ModuleInitialized := TRUE, subequently all subitems will be called to be initialized*)
METHOD Initializing
ModuleInitialized := TRUE;
END_METHOD

METHOD OnCyclicCall
END_METHOD

END_FUNCTION_BLOCK

// ---- _Mockups/Visitors/StringCollection.TcPOU
FUNCTION_BLOCK StringCollection
VAR_GENERIC CONSTANT
	StringMax : UDINT := 100;
END_VAR IMPLEMENTS I_StringCollection;
VAR
	Collection : ARRAY[0..StringMax] OF T_MaxString;
	_Entries   : UDINT;
END_VAR

METHOD AddString
VAR_INPUT
	StringToAdd : T_MaxString;
END_VAR
IF _Entries > StringMax THEN
	RETURN;
END_IF

Collection[_Entries] := StringToAdd;
_Entries			 := _Entries + 1;
END_METHOD

METHOD Clear : BOOL
VAR_INPUT
END_VAR
MEMSET(ADR(Collection), 0, SIZEOF(Collection));
_Entries := 0;
END_METHOD

PROPERTY Entries : UDINT
GET
Entries := _Entries;
END_GET
END_PROPERTY

END_FUNCTION_BLOCK

// ---- _Mockups/Visitors/ComponentVisitor_Mockup.TcPOU
FUNCTION_BLOCK ComponentVisitor_Mockup IMPLEMENTS I_ComponentVisitor
VAR
	StringCollection : I_StringCollection;
END_VAR

//FB_Init is always available implicitly and it is used primarily for initialization.

//The return value is not evaluated. For a specific influence, you can also declare the

//methods explicitly and provide additional code there with the standard initialization

//code. You can evaluate the return value.
METHOD FB_Init : BOOL
VAR_INPUT
	bInitRetains	 : BOOL; // TRUE: the retain variables are initialized (reset warm / reset cold)
	bInCopyCode		 : BOOL; // TRUE: the instance will be copied to the copy code afterward (online change)   
	StringCollection : I_StringCollection;
END_VAR
THIS^.StringCollection := StringCollection;
END_METHOD

METHOD VisitComponent
VAR_INPUT
	Component : I_Component;
END_VAR
StringCollection.AddString(Component.Name);
END_METHOD

END_FUNCTION_BLOCK

// ---- _Mockups/Modules/MachineModule_Mockup.TcPOU
FUNCTION_BLOCK MachineModule_Mockup EXTENDS Module
VAR
	SubModule				  : I_Module;
	TestComponent1			  : I_Component;
	TestComponent2			  : I_Component;
	StringCollection		  : StringCollection<100>;
	MachineModuleVisitor	  : GetSystemTreeNamesVisitor(StringCollection);
	QueryInterfaceResettables : QueryInterfaceResettables();
END_VAR

//FB_Init is always available implicitly and it is used primarily for initialization.

//The return value is not evaluated. For a specific influence, you can also declare the

//methods explicitly and provide additional code there with the standard initialization

//code. You can evaluate the return value.
METHOD FB_Init : BOOL
VAR_INPUT
	bInitRetains   : BOOL; // TRUE: the retain variables are initialized (reset warm / reset cold)
	bInCopyCode	   : BOOL; // TRUE: the instance will be copied to the copy code afterward (online change)   
	Name		   : T_MaxString;
	SubModule	   : I_Module;
	TestComponent1 : I_Component;
	TestComponent2 : I_Component;
END_VAR
THIS^.SubModule		 := SubModule;
THIS^.TestComponent1 := TestComponent1;
THIS^.TestComponent2 := TestComponent2;
SubModule.RegisterWithParent(THIS^);
TestComponent1.RegisterWithParent(THIS^);
TestComponent2.RegisterWithParent(THIS^);
END_METHOD

METHOD GetModuleByName : I_Module
VAR_INPUT
	Module : T_MaxString;
END_VAR
GetModuleByName := ModuleCollection.GetModuleByName(Module);
END_METHOD

(* This Module will be done initializeing when ModuleInitialized := TRUE;, subequently all subitems will be called to be initialized*)
METHOD Initializing
ModuleInitialized := TRUE;
END_METHOD

METHOD OnCyclicCall
MachineModuleVisitor.GetTree(THIS^);
QueryInterfaceResettables.GetAllResetComponents(THIS^);
END_METHOD

END_FUNCTION_BLOCK

// ---- _Mockups/Visitors/GetSystemTreeNamesVisitor.TcPOU
FUNCTION_BLOCK GetSystemTreeNamesVisitor IMPLEMENTS I_ModuleVisitor, I_ComponentVisitor
VAR
	StringCollection : I_StringCollection;
	Module			 : I_Module;
	Layer			 : STRING;
END_VAR

METHOD Clear
VAR_INPUT
END_VAR
StringCollection.Clear();
END_METHOD

//FB_Init is always available implicitly and it is used primarily for initialization.

//The return value is not evaluated. For a specific influence, you can also declare the

//methods explicitly and provide additional code there with the standard initialization

//code. You can evaluate the return value.
METHOD FB_Init : BOOL
VAR_INPUT
	bInitRetains	 : BOOL; // TRUE: the retain variables are initialized (reset warm / reset cold)
	bInCopyCode		 : BOOL; // TRUE: the instance will be copied to the copy code afterward (online change)   
	StringCollection : I_StringCollection;
END_VAR
THIS^.StringCollection := StringCollection;
END_METHOD

METHOD GetTree
VAR_INPUT
	EntryModule : I_Module;
END_VAR
IF EntryModule = 0 THEN
	RETURN;
END_IF

Module := EntryModule;
Clear();
StringCollection.AddString(Module.Name);
Layer := Module.Name;
Module.Components.Accept(THIS^);
Module.Modules.Accept(THIS^);
END_METHOD

METHOD VisitComponent
VAR_INPUT
	Component : I_Component;
END_VAR
StringCollection.AddString(CONCAT(Layer, CONCAT(' - ', Component.Name)));
END_METHOD

METHOD VisitModule
VAR_INPUT
	Module : I_Module;
END_VAR
StringCollection.AddString(Module.Name);
Layer := CONCAT(Layer, CONCAT(' - ', Module.Name));
Module.Components.Accept(THIS^);
Module.Modules.Accept(THIS^);
END_METHOD

END_FUNCTION_BLOCK

// ---- _Mockups/Visitors/QueryInterfaceResettables.TcPOU
FUNCTION_BLOCK QueryInterfaceResettables IMPLEMENTS I_ComponentVisitor
VAR
	Reset	   : ARRAY[0..10] OF I_Resettable;
	ResetCount : DINT;
END_VAR

METHOD GetAllResetComponents
VAR_INPUT
	EntryModule : I_Module;
END_VAR
ResetCount := 0;
EntryModule.Components.Accept(THIS^);
END_METHOD

METHOD VisitComponent
VAR_INPUT
	Component : I_Component;
END_VAR
IF __QUERYINTERFACE(Component, Reset[ResetCount]) THEN
	ResetCount := ResetCount + 1;
END_IF
END_METHOD

END_FUNCTION_BLOCK

// ---- _Mockups/Visitors/ModuleVisitor_Mockup.TcPOU
FUNCTION_BLOCK ModuleVisitor_Mockup IMPLEMENTS I_ModuleVisitor
VAR
	StringCollection : I_StringCollection;
END_VAR

//FB_Init is always available implicitly and it is used primarily for initialization.

//The return value is not evaluated. For a specific influence, you can also declare the

//methods explicitly and provide additional code there with the standard initialization

//code. You can evaluate the return value.
METHOD FB_Init : BOOL
VAR_INPUT
	bInitRetains	 : BOOL; // TRUE: the retain variables are initialized (reset warm / reset cold)
	bInCopyCode		 : BOOL; // TRUE: the instance will be copied to the copy code afterward (online change)   
	StringCollection : I_StringCollection;
END_VAR
THIS^.StringCollection := StringCollection;
END_METHOD

METHOD VisitModule
VAR_INPUT
	Module : I_Module;
END_VAR
StringCollection.AddString(Module.Name);
END_METHOD

END_FUNCTION_BLOCK

// ---- UnitTests/CyclicComponent/CyclicComponent_TEST.TcPOU
FUNCTION_BLOCK CyclicComponent_TEST
VAR
END_VAR

AcceptVisitor();
NameAssigned();
RegisterWithParent();
RegisterWithParent();
RegisterCyclic();
DeregisterWithParent();

METHOD AcceptVisitor
VAR_INST
	Expected : DINT;
	Actual	 : DINT;
END_VAR
VAR
	Component		 : CyclicComponent_Mockup('Component');
	StringCollection : StringCollection<100>;
	ComponentVisitor : ComponentVisitor_Mockup(StringCollection);
END_VAR
IF TestSuite.Test(__POUNAME()).ExecuteTest() THEN
	Expected := 1;
	Component.Accept(ComponentVisitor);
	Actual := StringCollection.Entries;
	TestSuite.Test(__POUNAME()).AssertEqual(Expected, Actual);
END_IF
END_METHOD

METHOD DeregisterWithParent
VAR_INST
	Expected : I_Component;
	Actual	 : I_Component;
END_VAR
VAR
	Component		 : CyclicComponent_Mockup('Component');
	StringCollection : StringCollection<100>;
	ComponentVisitor : ComponentVisitor_Mockup(StringCollection);
	Module			 : EquipmentModule_Mockup('Module', Component, Component);
END_VAR
IF TestSuite.Test(__POUNAME()).ExecuteTest() THEN
	Expected := 0;
	Component.DeregisterWithParent(Module);
	Component.DeregisterWithParent(Module);
	Actual := Module.GetComponentByName('Component');
	TestSuite.Test(__POUNAME()).AssertEqual(Expected, Actual);
END_IF
END_METHOD

METHOD NameAssigned
VAR_INST
	Expected : STRING;
	Actual	 : STRING;
END_VAR
VAR
	Component		 : CyclicComponent_Mockup('Component');
	StringCollection : StringCollection<100>;
	ComponentVisitor : ComponentVisitor_Mockup(StringCollection);
END_VAR
IF TestSuite.Test(__POUNAME()).ExecuteTest() THEN
	Expected := 'Component';
	Actual	 := Component.Name;
	TestSuite.Test(__POUNAME()).AssertEqual(Expected, Actual);
END_IF
END_METHOD

METHOD RegisterCyclic
VAR_INST
	Expected : BOOL;
	Actual	 : BOOL;
END_VAR
VAR
	Component		 : CyclicComponent_Mockup('Component');
	StringCollection : StringCollection<100>;
	ComponentVisitor : ComponentVisitor_Mockup(StringCollection);
	Module	: EquipmentModule_Mockup('Module', Component, Component);
END_VAR
IF TestSuite.Test(__POUNAME()).ExecuteTest() THEN
	Expected := TRUE;
	Module.CyclicLogic();
	Actual := Component.WasCalled;
	TestSuite.Test(__POUNAME()).AssertEqual(Expected, Actual);
END_IF
END_METHOD

METHOD RegisterWithParent
VAR_INST
	Expected : STRING;
	Actual	 : STRING;
END_VAR
VAR
	Component		 : CyclicComponent_Mockup('Component');
	StringCollection : StringCollection<100>;
	ComponentVisitor : ComponentVisitor_Mockup(StringCollection);
	Module	: EquipmentModule_Mockup('Module', Component, Component);
END_VAR
IF TestSuite.Test(__POUNAME()).ExecuteTest() THEN
	Expected := 'Component';
	Actual	 := Module.GetComponentByName('Component').Name;
	TestSuite.Test(__POUNAME()).AssertEqual(Expected, Actual);
END_IF
END_METHOD

END_FUNCTION_BLOCK

// ---- UnitTests/Component/Component_TEST.TcPOU
FUNCTION_BLOCK Component_TEST
VAR
END_VAR

AcceptVisitor();
NameAssigned();
RegisterWithParent();
DeregisterWithParent();

METHOD AcceptVisitor
VAR_INST
	Expected : DINT;
	Actual	 : DINT;
END_VAR
VAR
	StringCollection : StringCollection<100>;
	ComponentVisitor : ComponentVisitor_Mockup(StringCollection);
	Component : Component_Mockup('Component');
END_VAR
IF TestSuite.Test(__POUNAME()).ExecuteTest() THEN
	Expected := 1;
	Component.Accept(ComponentVisitor);
	Actual := StringCollection.Entries;
	TestSuite.Test(__POUNAME()).AssertEqual(Expected, Actual);
END_IF
END_METHOD

METHOD DeregisterWithParent
VAR_INST
	Expected : I_Component;
	Actual	 : I_Component;
END_VAR
VAR
	Component : Component_Mockup('Component');
	Module	: EquipmentModule_Mockup('Module', Component, Component);
END_VAR
IF TestSuite.Test(__POUNAME()).ExecuteTest() THEN
	Expected := 0;
	Component.DeregisterWithParent(Module);
	Component.DeregisterWithParent(Module);
	Actual := Module.GetComponentByName('Component');
	TestSuite.Test(__POUNAME()).AssertEqual(Expected, Actual);
END_IF
END_METHOD

METHOD NameAssigned
VAR_INST
	Expected : STRING;
	Actual	 : STRING;
END_VAR
VAR
	StringCollection : StringCollection<100>;
	ComponentVisitor : ComponentVisitor_Mockup(StringCollection);
	Component : Component_Mockup('Component');
END_VAR
IF TestSuite.Test(__POUNAME()).ExecuteTest() THEN
	Expected := 'Component';
	Actual	 := Component.Name;
	TestSuite.Test(__POUNAME()).AssertEqual(Expected, Actual);
END_IF
END_METHOD

METHOD RegisterWithParent
VAR_INST
	Expected : STRING;
	Actual	 : STRING;
END_VAR
VAR
	Component : Component_Mockup('Component');
	Module	: EquipmentModule_Mockup('Module', Component, Component);
END_VAR
IF TestSuite.Test(__POUNAME()).ExecuteTest() THEN
	Expected := 'Component';
	Actual	 := Module.GetComponentByName('Component').Name;
	TestSuite.Test(__POUNAME()).AssertEqual(Expected, Actual);
END_IF
END_METHOD

END_FUNCTION_BLOCK

// ---- _Mockups/Components/Component_Mockup.TcPOU
FUNCTION_BLOCK Component_Mockup EXTENDS Component
VAR
END_VAR

END_FUNCTION_BLOCK

// ---- UnitTests/ModuleCollection/ModuleCollection_TEST.TcPOU
FUNCTION_BLOCK ModuleCollection_TEST
VAR

END_VAR

CollectionAddsModuleSucessfully();
CollectionRejectsAddingModuleDuplicate();
CollectionRejectsAddingNullModule();
CollectionRejectsAddingTooManyModules();
CollectionRejectsRemoveWhenEmpty();
CollectionRejectsRemoveWhenNotFound();
CollectionRejectsRemovingNullModule();
CollectionRemovesModuleSuccessfully();
GetModuleByName();
CollectionGetItemAtIndex();
CollectionGetCount();

METHOD CollectionAddsModuleSucessfully
VAR
	Expected	: BOOL := TRUE;
	Actual		: BOOL;
	Module			 : Module_Mockup('Mockup Module');
	ModuleCollection : ModuleCollection<ApplicationBaseParameter.MaxCountInCollections>;
END_VAR
IF TestSuite.Test(__POUNAME()).ExecuteTest() THEN
	Actual := ModuleCollection.AddModule(Module) = RegistrationResult.Succeeded;
	TestSuite.Test(__POUNAME()).AssertEqual(Expected, Actual);
END_IF
END_METHOD

METHOD CollectionGetCount
VAR
	Expected		 : UDINT;
	Actual			 : UDINT;
	ModuleCollection : ModuleCollection<ApplicationBaseParameter.MaxCountInCollections>;
	Module1			 : Module_Mockup('Mockup Module 1');
END_VAR
IF TestSuite.Test(__POUNAME()).ExecuteTest() THEN
	Expected := 1;
	ModuleCollection.AddModule(Module1);
	Actual := ModuleCollection.Count;
	TestSuite.Test(__POUNAME()).AssertEqual(Expected, Actual);
END_IF
END_METHOD

METHOD CollectionGetItemAtIndex
VAR
	Expected		 : BOOL := TRUE;
	Actual			 : BOOL;
	ModuleCollection : ModuleCollection<2>;
	Module1			 : Module_Mockup('Mockup Module 1');
	Module2			 : Module_Mockup('Mockup Module 2');
	ReturnedModule	 : I_Module;
END_VAR
IF TestSuite.Test(__POUNAME()).ExecuteTest() THEN
	ModuleCollection.AddModule(Module1);
	ModuleCollection.AddModule(Module2);
	ReturnedModule := ModuleCollection.GetAtIndex(1);
	Actual		   := ReturnedModule.Name = Module2.Name;
	TestSuite.Test(__POUNAME()).AssertEqual(Expected, Actual);
END_IF
END_METHOD

METHOD CollectionRejectsAddingModuleDuplicate
VAR
	Expected	: BOOL := TRUE;
	Actual		: BOOL;
	Module			 : Module_Mockup('Mockup Module');
	ModuleCollection : ModuleCollection<ApplicationBaseParameter.MaxCountInCollections>;
END_VAR
IF TestSuite.Test(__POUNAME()).ExecuteTest() THEN
	ModuleCollection.AddModule(Module);
	Actual := ModuleCollection.AddModule(Module) = RegistrationResult.AlreadyAdded;
	TestSuite.Test(__POUNAME()).AssertEqual(Expected, Actual);
END_IF
END_METHOD

METHOD CollectionRejectsAddingNullModule
VAR
	Expected	: BOOL := TRUE;
	Actual		: BOOL;
	ModuleCollection : ModuleCollection<ApplicationBaseParameter.MaxCountInCollections>;
END_VAR
IF TestSuite.Test(__POUNAME()).ExecuteTest() THEN
	Actual := ModuleCollection.AddModule(16#0) = RegistrationResult.NullReference;
	TestSuite.Test(__POUNAME()).AssertEqual(Expected, Actual);
END_IF
END_METHOD

METHOD CollectionRejectsAddingTooManyModules
VAR
	Expected	: BOOL := TRUE;
	Actual		: BOOL;
	Module1			 : Module_Mockup('Mockup Module');
	Module2			 : Module_Mockup('Mockup Module');
	ModuleCollection : ModuleCollection<1>;
END_VAR
IF TestSuite.Test(__POUNAME()).ExecuteTest() THEN
	ModuleCollection.AddModule(Module1);
	Actual := ModuleCollection.AddModule(Module2) = RegistrationResult.TooManyComponents;
	TestSuite.Test(__POUNAME()).AssertEqual(Expected, Actual);
END_IF
END_METHOD

METHOD CollectionRejectsRemoveWhenEmpty
VAR
	Expected	: BOOL := TRUE;
	Actual		: BOOL;
	Module			 : Module_Mockup('Mockup Module');
	ModuleCollection : ModuleCollection<ApplicationBaseParameter.MaxCountInCollections>;
END_VAR
IF TestSuite.Test(__POUNAME()).ExecuteTest() THEN
	Actual := ModuleCollection.RemoveModule(Module) = RegistrationResult.CollectionEmpty;
	TestSuite.Test(__POUNAME()).AssertEqual(Expected, Actual);
END_IF
END_METHOD

METHOD CollectionRejectsRemoveWhenNotFound
VAR
	Expected	: BOOL := TRUE;
	Actual		: BOOL;
	Module1			 : Module_Mockup('Mockup Module');
	Module2			 : Module_Mockup('Mockup Module');
	ModuleCollection : ModuleCollection<ApplicationBaseParameter.MaxCountInCollections>;
END_VAR
IF TestSuite.Test(__POUNAME()).ExecuteTest() THEN
	ModuleCollection.AddModule(Module1);
	Actual := ModuleCollection.RemoveModule(Module2) = RegistrationResult.NotFoundInCollection;
	TestSuite.Test(__POUNAME()).AssertEqual(Expected, Actual);
END_IF
END_METHOD

METHOD CollectionRejectsRemovingNullModule
VAR
	Expected	: BOOL := TRUE;
	Actual		: BOOL;
	ModuleCollection : ModuleCollection<ApplicationBaseParameter.MaxCountInCollections>;
END_VAR
IF TestSuite.Test(__POUNAME()).ExecuteTest() THEN
	Actual := ModuleCollection.RemoveModule(16#0) = RegistrationResult.NullReference;
	TestSuite.Test(__POUNAME()).AssertEqual(Expected, Actual);
END_IF
END_METHOD

METHOD CollectionRemovesModuleSuccessfully
VAR
	Expected	: BOOL := TRUE;
	Actual		: BOOL;
	Module			 : Module_Mockup('Mockup Module');
	ModuleCollection : ModuleCollection<ApplicationBaseParameter.MaxCountInCollections>;
	AddedModule : I_Module := Module;
	CollectionModule : I_Module;
END_VAR
IF TestSuite.Test(__POUNAME()).ExecuteTest() THEN
	ModuleCollection.AddModule(Module);
	Actual := ModuleCollection.RemoveModule(Module) = RegistrationResult.Succeeded;
	TestSuite.Test(__POUNAME()).AssertEqual(Expected, Actual);
END_IF
END_METHOD

METHOD GetModuleByName
VAR
	Expected	: STRING;
	Actual		: STRING;
	BaseModule	: I_Module;
	AddedModule : I_Module;
	Module			 : Module_Mockup('Mockup Module');
	ModuleCollection : ModuleCollection<ApplicationBaseParameter.MaxCountInCollections>;
END_VAR
IF TestSuite.Test(__POUNAME()).ExecuteTest() THEN
	Expected   := 'Mockup Module';
	BaseModule := Module;
	ModuleCollection.AddModule(Module);
	AddedModule := ModuleCollection.GetModuleByName(Expected);
	Actual		:= AddedModule.Name;
	TestSuite.Test(__POUNAME()).AssertEqual(Expected, Actual);
END_IF
END_METHOD

END_FUNCTION_BLOCK

// ---- UnitTests/Tracing/Tracing_TEST.TcPOU
FUNCTION_BLOCK Tracing_TEST
VAR
	i : DINT;
END_VAR

TcTraceLogMessageSent();
AdsTraceLogSent();
TraceLogAcceptsCritical();
TraceLogAcceptsError();
TraceLogAcceptsWarning();
TraceLogAcceptsInfo();
TraceLogAcceptsVerbose();
TraceLogRejectsCriticalTracingOff();
TraceLogRejectsErrorTracingLvlHigh();
TraceLogRejectsErrorTracingOff();
TraceLogRejectsWarningTracingLvlHigh();
TraceLogRejectsWarningTracingOff();
TraceLogRejectsInfoTracingLvlHigh();
TraceLogRejectsInfoTracingOff();
TraceLogRejectsVerboseTracingLvlHigh();
TraceLogRejectsVerboseTracingOff();

METHOD AdsTraceLogSent
VAR
	Expected : DINT;
	Actual	 : DINT;
END_VAR
IF TestSuite.Test(__POUNAME()).ExecuteTest() THEN
	Expected := 2;
	Trace.LogMessage('Test', 'Message Ads Logger');
	Actual := CoreTrace.AdsLogger.MessagesThisScan;
	TestSuite.Test(__POUNAME()).AssertEqual(Expected, Actual);
END_IF
END_METHOD

METHOD TcTraceLogMessageSent
VAR
	Expected : DINT;
	Actual	 : DINT;
END_VAR
IF TestSuite.Test(__POUNAME()).ExecuteTest() THEN
	Expected := 1;
	Trace.LogMessage('Test', 'Message TcEvent');
	Actual := CoreTrace.TcEventLogger.MessagesThisScan;
	TestSuite.Test(__POUNAME()).AssertEqual(Expected, Actual);
END_IF
END_METHOD

METHOD TraceLogAcceptsCritical
VAR
	Expected : DINT;
	Actual	 : DINT;
END_VAR
IF TestSuite.Test(__POUNAME()).ExecuteTest() THEN
	Trace.TraceLevel := TcEventSeverityExt.Verbose;
	Expected := CoreTrace.AdsLogger.MessagesThisScan + 1;
	Trace.Critical('Test', 'Message TcEvent');
	Actual := CoreTrace.AdsLogger.MessagesThisScan;
	TestSuite.Test(__POUNAME()).AssertEqual(Expected, Actual);
END_IF
END_METHOD

METHOD TraceLogAcceptsError
VAR
	Expected : DINT;
	Actual	 : DINT;
END_VAR
IF TestSuite.Test(__POUNAME()).ExecuteTest() THEN
	Trace.TraceLevel := TcEventSeverityExt.Verbose;
	Expected := CoreTrace.AdsLogger.MessagesThisScan + 1;
	Trace.Error('Test', 'Message TcEvent');
	Actual := CoreTrace.AdsLogger.MessagesThisScan;
	TestSuite.Test(__POUNAME()).AssertEqual(Expected, Actual);
END_IF
END_METHOD

METHOD TraceLogAcceptsInfo
VAR
	Expected : DINT;
	Actual	 : DINT;
END_VAR
IF TestSuite.Test(__POUNAME()).ExecuteTest() THEN
	Trace.TraceLevel := TcEventSeverityExt.Verbose;
	Expected := CoreTrace.AdsLogger.MessagesThisScan + 1;
	Trace.Info('Test', 'Message TcEvent');
	Actual := CoreTrace.AdsLogger.MessagesThisScan;
	TestSuite.Test(__POUNAME()).AssertEqual(Expected, Actual);
END_IF
END_METHOD

METHOD TraceLogAcceptsVerbose
VAR
	Expected : DINT;
	Actual	 : DINT;
END_VAR
IF TestSuite.Test(__POUNAME()).ExecuteTest() THEN
	Trace.TraceLevel := TcEventSeverityExt.Verbose;
	Expected := CoreTrace.AdsLogger.MessagesThisScan + 1;
	Trace.Verbose('Test', 'Message TcEvent');
	Actual := CoreTrace.AdsLogger.MessagesThisScan;
	TestSuite.Test(__POUNAME()).AssertEqual(Expected, Actual);
END_IF
END_METHOD

METHOD TraceLogAcceptsWarning
VAR
	Expected : DINT;
	Actual	 : DINT;
END_VAR
IF TestSuite.Test(__POUNAME()).ExecuteTest() THEN
	Trace.TraceLevel := TcEventSeverityExt.Verbose;
	Expected := CoreTrace.AdsLogger.MessagesThisScan + 1;
	Trace.Warning('Test', 'Message TcEvent');
	Actual := CoreTrace.AdsLogger.MessagesThisScan;
	TestSuite.Test(__POUNAME()).AssertEqual(Expected, Actual);
END_IF
END_METHOD

METHOD TraceLogRejectsCriticalTracingOff
VAR
	Expected : DINT;
	Actual	 : DINT;
END_VAR
IF TestSuite.Test(__POUNAME()).ExecuteTest() THEN
	Trace.TraceLevel := TcEventSeverityExt.Off;
	Expected := CoreTrace.AdsLogger.MessagesThisScan;
	Trace.Critical('Test', 'Message TcEvent');
	Actual := CoreTrace.AdsLogger.MessagesThisScan;
	TestSuite.Test(__POUNAME()).AssertEqual(Expected, Actual);
END_IF
END_METHOD

METHOD TraceLogRejectsErrorTracingLvlHigh
VAR
	Expected : DINT;
	Actual	 : DINT;
END_VAR
IF TestSuite.Test(__POUNAME()).ExecuteTest() THEN
	Trace.TraceLevel := TcEventSeverityExt.Critical;
	Expected := CoreTrace.AdsLogger.MessagesThisScan;
	Trace.Error('Test', 'Message TcEvent');
	Actual := CoreTrace.AdsLogger.MessagesThisScan;
	TestSuite.Test(__POUNAME()).AssertEqual(Expected, Actual);
END_IF
END_METHOD

METHOD TraceLogRejectsErrorTracingOff
VAR
	Expected : DINT;
	Actual	 : DINT;
END_VAR
IF TestSuite.Test(__POUNAME()).ExecuteTest() THEN
	Trace.TraceLevel := TcEventSeverityExt.Off;
	Expected := CoreTrace.AdsLogger.MessagesThisScan;
	Trace.Error('Test', 'Message TcEvent');
	Actual := CoreTrace.AdsLogger.MessagesThisScan;
	TestSuite.Test(__POUNAME()).AssertEqual(Expected, Actual);
END_IF
END_METHOD

METHOD TraceLogRejectsInfoTracingLvlHigh
VAR
	Expected : DINT;
	Actual	 : DINT;
END_VAR
IF TestSuite.Test(__POUNAME()).ExecuteTest() THEN
	Trace.TraceLevel := TcEventSeverityExt.Warning;
	Expected := CoreTrace.AdsLogger.MessagesThisScan;
	Trace.Info('Test', 'Message TcEvent');
	Actual := CoreTrace.AdsLogger.MessagesThisScan;
	TestSuite.Test(__POUNAME()).AssertEqual(Expected, Actual);
END_IF
END_METHOD

METHOD TraceLogRejectsInfoTracingOff
VAR
	Expected : DINT;
	Actual	 : DINT;
END_VAR
IF TestSuite.Test(__POUNAME()).ExecuteTest() THEN
	Trace.TraceLevel := TcEventSeverityExt.Off;
	Expected := CoreTrace.AdsLogger.MessagesThisScan;
	Trace.Info('Test', 'Message TcEvent');
	Actual := CoreTrace.AdsLogger.MessagesThisScan;
	TestSuite.Test(__POUNAME()).AssertEqual(Expected, Actual);
END_IF
END_METHOD

METHOD TraceLogRejectsVerboseTracingLvlHigh
VAR
	Expected : DINT;
	Actual	 : DINT;
END_VAR
IF TestSuite.Test(__POUNAME()).ExecuteTest() THEN
	Trace.TraceLevel := TcEventSeverityExt.Info;
	Expected := CoreTrace.AdsLogger.MessagesThisScan;
	Trace.Verbose('Test', 'Message TcEvent');
	Actual := CoreTrace.AdsLogger.MessagesThisScan;
	TestSuite.Test(__POUNAME()).AssertEqual(Expected, Actual);
END_IF
END_METHOD

METHOD TraceLogRejectsVerboseTracingOff
VAR
	Expected : DINT;
	Actual	 : DINT;
END_VAR
IF TestSuite.Test(__POUNAME()).ExecuteTest() THEN
	Trace.TraceLevel := TcEventSeverityExt.Off;
	Expected := CoreTrace.AdsLogger.MessagesThisScan;
	Trace.Verbose('Test', 'Message TcEvent');
	Actual := CoreTrace.AdsLogger.MessagesThisScan;
	TestSuite.Test(__POUNAME()).AssertEqual(Expected, Actual);
END_IF
END_METHOD

METHOD TraceLogRejectsWarningTracingLvlHigh
VAR
	Expected : DINT;
	Actual	 : DINT;
END_VAR
IF TestSuite.Test(__POUNAME()).ExecuteTest() THEN
	Trace.TraceLevel := TcEventSeverityExt.Error;
	Expected := CoreTrace.AdsLogger.MessagesThisScan;
	Trace.Warning('Test', 'Message TcEvent');
	Actual := CoreTrace.AdsLogger.MessagesThisScan;
	TestSuite.Test(__POUNAME()).AssertEqual(Expected, Actual);
END_IF
END_METHOD

METHOD TraceLogRejectsWarningTracingOff
VAR
	Expected : DINT;
	Actual	 : DINT;
END_VAR
IF TestSuite.Test(__POUNAME()).ExecuteTest() THEN
	Trace.TraceLevel := TcEventSeverityExt.Off;
	Expected := CoreTrace.AdsLogger.MessagesThisScan;
	Trace.Warning('Test', 'Message TcEvent');
	Actual := CoreTrace.AdsLogger.MessagesThisScan;
	TestSuite.Test(__POUNAME()).AssertEqual(Expected, Actual);
END_IF
END_METHOD

END_FUNCTION_BLOCK

// ---- UnitTests/Initializer/Initializer_TEST.TcPOU
FUNCTION_BLOCK Initializer_TEST
VAR
END_VAR

CollectionAddsInitSucessfully();
CollectionRejectsAddingInitDuplicate();
CollectionRejectsAddingNullInit();
CollectionRejectsAddingTooManyInits();
CollectionRejectsRemoveWhenEmpty();
CollectionRejectsRemoveWhenNotFound();
CollectionRejectsRemovingNullInit();
CollectionRemovesInitSuccessfully();
FeedbackAllSubItemsInitializedFalse();
FeedbackAllSubItemsInitializedTrue();

METHOD CollectionAddsInitSucessfully
VAR
	Expected	   : BOOL := TRUE;
	Actual		   : BOOL;
	CyclicRunner : CyclicRunner<ApplicationBaseParameter.MaxCountInCollections>;
	Cyclic	 : CyclicComponent_Mockup(Name := 'Cyclic 1');
END_VAR
IF TestSuite.Test(__POUNAME()).ExecuteTest() THEN
	Actual := CyclicRunner.AddCallee(Cyclic) = RegistrationResult.Succeeded;
	TestSuite.Test(__POUNAME()).AssertEqual(Expected, Actual);
END_IF
END_METHOD

METHOD CollectionRejectsAddingInitDuplicate
VAR
	Expected : BOOL := TRUE;
	Actual	 : BOOL;
	Initializer : Initializer<ApplicationBaseParameter.MaxCountInCollections>;
	Init	: InitializableComponent_Mockup(Name := 'Component 1');
END_VAR
IF TestSuite.Test(__POUNAME()).ExecuteTest() THEN
	Initializer.AddInitialize(Init);
	Actual := Initializer.AddInitialize(Init) = RegistrationResult.AlreadyAdded;
	TestSuite.Test(__POUNAME()).AssertEqual(Expected, Actual);
END_IF
END_METHOD

METHOD CollectionRejectsAddingNullInit
VAR
	Expected : BOOL := TRUE;
	Actual	 : BOOL;
	Initializer : Initializer<ApplicationBaseParameter.MaxCountInCollections>;
	Init	: InitializableComponent_Mockup(Name := 'Component 1');
END_VAR
IF TestSuite.Test(__POUNAME()).ExecuteTest() THEN
	Actual := Initializer.AddInitialize(16#0) = RegistrationResult.NullReference;
	TestSuite.Test(__POUNAME()).AssertEqual(Expected, Actual);
END_IF
END_METHOD

METHOD CollectionRejectsAddingTooManyInits
VAR
	Expected : BOOL := TRUE;
	Actual	 : BOOL;
	Initializer : Initializer<1>;
	Init1	: InitializableComponent_Mockup(Name := 'Component 1');
	Init2	: InitializableComponent_Mockup(Name := 'Component 1');
END_VAR
IF TestSuite.Test(__POUNAME()).ExecuteTest() THEN
	Initializer.AddInitialize(Init1);
	Actual := Initializer.AddInitialize(Init2) = RegistrationResult.TooManyComponents;
	TestSuite.Test(__POUNAME()).AssertEqual(Expected, Actual);
END_IF
END_METHOD

METHOD CollectionRejectsRemoveWhenEmpty
VAR
	Expected : BOOL := TRUE;
	Actual	 : BOOL;
	Initializer : Initializer<ApplicationBaseParameter.MaxCountInCollections>;
	Init	: InitializableComponent_Mockup(Name := 'Component 1');
END_VAR
IF TestSuite.Test(__POUNAME()).ExecuteTest() THEN
	Actual := Initializer.RemoveInitialize(Init) = RegistrationResult.CollectionEmpty;
	TestSuite.Test(__POUNAME()).AssertEqual(Expected, Actual);
END_IF
END_METHOD

METHOD CollectionRejectsRemoveWhenNotFound
VAR
	Expected : BOOL := TRUE;
	Actual	 : BOOL;
	Initializer : Initializer<ApplicationBaseParameter.MaxCountInCollections>;
	Init1	: InitializableComponent_Mockup(Name := 'Component 1');
	Init2	: InitializableComponent_Mockup(Name := 'Component 1');
END_VAR
IF TestSuite.Test(__POUNAME()).ExecuteTest() THEN
	Initializer.AddInitialize(Init1);
	Actual := Initializer.RemoveInitialize(Init2) = RegistrationResult.NotFoundInCollection;
	TestSuite.Test(__POUNAME()).AssertEqual(Expected, Actual);
END_IF
END_METHOD

METHOD CollectionRejectsRemovingNullInit
VAR
	Expected : BOOL := TRUE;
	Actual	 : BOOL;
	Initializer : Initializer<ApplicationBaseParameter.MaxCountInCollections>;
END_VAR
IF TestSuite.Test(__POUNAME()).ExecuteTest() THEN
	Actual := Initializer.RemoveInitialize(16#0) = RegistrationResult.NullReference;
	TestSuite.Test(__POUNAME()).AssertEqual(Expected, Actual);
END_IF
END_METHOD

METHOD CollectionRemovesInitSuccessfully
VAR
	Expected : BOOL := TRUE;
	Actual	 : BOOL;
	Initializer : Initializer<ApplicationBaseParameter.MaxCountInCollections>;
	Init	: InitializableComponent_Mockup(Name := 'Component 1');
	AddedCyclic : I_Initializable := Init;
	CollectionInit : I_Initializable;
END_VAR
IF TestSuite.Test(__POUNAME()).ExecuteTest() THEN
	Initializer.AddInitialize(Init);
	Actual := Initializer.RemoveInitialize(Init) = RegistrationResult.Succeeded;
	TestSuite.Test(__POUNAME()).AssertEqual(Expected, Actual);
END_IF
END_METHOD

METHOD FeedbackAllSubItemsInitializedFalse
VAR_INST
	Expected : BOOL;
	Actual	 : BOOL;
END_VAR
VAR
	Initializer : Initializer<ApplicationBaseParameter.MaxCountInCollections>;
	Component1	: InitializableComponent_Mockup(Name := 'Component 1');
	Component2	: InitializableComponent_Mockup(Name := 'Component 1');
	Component3	: InitializableComponent_Mockup(Name := 'Component 1');
END_VAR
IF TestSuite.Test(__POUNAME()).ExecuteTest() THEN
	Expected := TRUE;
	Initializer.AddInitialize(Component1);
	Initializer.AddInitialize(Component2);
	Initializer.AddInitialize(Component3);
	Initializer.Initializing();
	Actual := Component1.InitializeWasCalled AND Component2.InitializeWasCalled AND Component3.InitializeWasCalled AND NOT Initializer.Initialized;
	TestSuite.Test(__POUNAME()).AssertEqual(Expected, Actual);
END_IF
END_METHOD

METHOD FeedbackAllSubItemsInitializedTrue
VAR_INST
	Expected : BOOL;
	Actual	 : BOOL;
END_VAR
VAR
	Initializer : Initializer<ApplicationBaseParameter.MaxCountInCollections>;
	Component1	: InitializableComponent_Mockup(Name := 'Component 1');
	Component2	: InitializableComponent_Mockup(Name := 'Component 1');
	Component3	: InitializableComponent_Mockup(Name := 'Component 1');
END_VAR
IF TestSuite.Test(__POUNAME()).ExecuteTest() THEN
	Expected			   := TRUE;
	Initializer.AddInitialize(Component1);
	Initializer.AddInitialize(Component2);
	Initializer.AddInitialize(Component3);
	Component1.Initialized := TRUE;
	Component2.Initialized := TRUE;
	Component3.Initialized := TRUE;
	Initializer.Initializing();
	Actual := Component1.InitializeWasCalled AND Component2.InitializeWasCalled AND Component3.InitializeWasCalled AND Initializer.Initialized;
	TestSuite.Test(__POUNAME()).AssertEqual(Expected, Actual);
END_IF
END_METHOD

END_FUNCTION_BLOCK

// ---- UnitTests/Events/Events_TEST.TcPOU
FUNCTION_BLOCK Events_TEST
VAR
	CyclicComponent_Mockup : CyclicComponent_Mockup('UnitTest Component');
	MockupComponentTcEvent : MockupComponentTcEvent('UnitTest Component Events', CyclicComponent_Mockup);
	Trigger				   : BOOL;
END_VAR

MockupComponentTcEvent.SetEventReactions(10,
										 20,
										 30,
										 40,
										 50);

RaiseVerboseEventAndCheckReaction();
RaiseInfoEventAndCheckReaction();
RaiseWarningEventAndCheckReaction();
RaiseErrorEventAndCheckReaction();
RaiseCriticalEventAndCheckReaction();
ClearEvents();
SetEventAndRaise();
CheckIsResettable();
Reset();

METHOD CheckIsResettable
VAR_INST
	Expected : BOOL;
	Actual	 : BOOL;
END_VAR
IF TestSuite.Test(__POUNAME()).ExecuteTest() THEN
	Expected := TRUE;
	Trigger := FALSE;
	MockupComponentTcEvent.Events.CyclicLogic();
	Actual := MockupComponentTcEvent.Events.IsResettable;
	TestSuite.Test(__POUNAME()).AssertEqual(Expected, Actual);
END_IF
END_METHOD

METHOD ClearEvents
VAR
	Expected : DINT;
	Actual	 : DINT;
END_VAR
IF TestSuite.Test(__POUNAME()).ExecuteTest() THEN
	Expected := 10;
	MockupComponentTcEvent.Reset();
	Actual := MockupComponentTcEvent.GetHighestActiveEventReaction();
	TestSuite.Test(__POUNAME()).AssertEqual(Expected, Actual);
END_IF
END_METHOD

METHOD RaiseCriticalEventAndCheckReaction
VAR
	Expected : DINT;
	Actual	 : DINT;
END_VAR
IF TestSuite.Test(__POUNAME()).ExecuteTest() THEN
	Expected := 50;
	MockupComponentTcEvent.RaiseTestEvent(TcEventSeverity.Critical);
	Actual := MockupComponentTcEvent.GetHighestActiveEventReaction();
	TestSuite.Test(__POUNAME()).AssertEqual(Expected, Actual);
END_IF
END_METHOD

METHOD RaiseErrorEventAndCheckReaction
VAR
	Expected : DINT;
	Actual	 : DINT;
END_VAR
IF TestSuite.Test(__POUNAME()).ExecuteTest() THEN
	Expected := 40;
	MockupComponentTcEvent.RaiseTestEvent(TcEventSeverity.Error);
	Actual := MockupComponentTcEvent.GetHighestActiveEventReaction();
	TestSuite.Test(__POUNAME()).AssertEqual(Expected, Actual);
END_IF
END_METHOD

METHOD RaiseInfoEventAndCheckReaction
VAR
	Expected : DINT;
	Actual	 : DINT;
END_VAR
IF TestSuite.Test(__POUNAME()).ExecuteTest() THEN
	Expected := 20;
	MockupComponentTcEvent.RaiseTestEvent(TcEventSeverity.Info);
	Actual := MockupComponentTcEvent.GetHighestActiveEventReaction();
	TestSuite.Test(__POUNAME()).AssertEqual(Expected, Actual);
END_IF
END_METHOD

METHOD RaiseVerboseEventAndCheckReaction
VAR
	Expected : DINT;
	Actual	 : DINT;
END_VAR
IF TestSuite.Test(__POUNAME()).ExecuteTest() THEN
	Expected := 10;
	MockupComponentTcEvent.RaiseTestEvent(TcEventSeverity.Verbose);
	Actual := MockupComponentTcEvent.GetHighestActiveEventReaction();
	TestSuite.Test(__POUNAME()).AssertEqual(Expected, Actual);
END_IF
END_METHOD

METHOD RaiseWarningEventAndCheckReaction
VAR
	Expected : DINT;
	Actual	 : DINT;
END_VAR
IF TestSuite.Test(__POUNAME()).ExecuteTest() THEN
	Expected := 30;
	MockupComponentTcEvent.RaiseTestEvent(TcEventSeverity.Warning);
	Actual := MockupComponentTcEvent.GetHighestActiveEventReaction();
	TestSuite.Test(__POUNAME()).AssertEqual(Expected, Actual);
END_IF
END_METHOD

METHOD Reset
VAR
	Expected : DINT;
	Actual	 : DINT;
END_VAR
IF TestSuite.Test(__POUNAME()).ExecuteTest() THEN
	Expected := 10;
	MockupComponentTcEvent.Reset();
	Actual := MockupComponentTcEvent.GetHighestActiveEventReaction();
	TestSuite.Test(__POUNAME()).AssertEqual(Expected, Actual);
END_IF
END_METHOD

METHOD SetEventAndRaise
VAR_INST
	Expected : DINT;
	Actual	 : DINT;
END_VAR
IF TestSuite.Test(__POUNAME()).ExecuteTest() THEN
	Expected := 40;
	MockupComponentTcEvent.Events.SetEvent(E_TestComponent.SetEvent, ADR(Trigger), FALSE);
	Trigger := TRUE;
	MockupComponentTcEvent.Events.CyclicLogic();
	Actual := MockupComponentTcEvent.GetHighestActiveEventReaction();
	TestSuite.Test(__POUNAME()).AssertEqual(Expected, Actual);
END_IF
END_METHOD

END_FUNCTION_BLOCK

// ---- _Mockups/Components/MockupComponentTcEvent.TcPOU
FUNCTION_BLOCK MockupComponentTcEvent EXTENDS Component IMPLEMENTS I_EventReaction
VAR
	Events : TcEventClass('');
END_VAR

//FB_Init is always available implicitly and it is used primarily for initialization.

//The return value is not evaluated. For a specific influence, you can also declare the

//methods explicitly and provide additional code there with the standard initialization

//code. You can evaluate the return value.
METHOD FB_Init : BOOL
VAR_INPUT
	bInitRetains : BOOL; // TRUE: the retain variables are initialized (reset warm / reset cold)
	bInCopyCode	 : BOOL; // TRUE: the instance will be copied to the copy code afterward (online change) 
	Name		 : T_MaxString;
	Component	 : I_Component;
END_VAR
Events.GenerateTcEvents(Component.Name, ADR(TC_Events.TestComponent), SIZEOF(ST_TestComponent));
END_METHOD

METHOD GetHighestActiveEventReaction : DINT
GetHighestActiveEventReaction := Events.GetHighestActiveEventReaction();
END_METHOD

METHOD GetHighestActiveEventSeverity : TcEventSeverity
GetHighestActiveEventSeverity := Events.GetHighestActiveEventSeverity();
END_METHOD

METHOD RaiseTestEvent
VAR_INPUT
	Severity : TcEventSeverity;
END_VAR
CASE Severity OF
	TcEventSeverity.Critical:
		Events.RaiseEvent(E_TestComponent.CriticalEvent);

	TcEventSeverity.Error:
		Events.RaiseEvent(E_TestComponent.ErrorEvent);

	TcEventSeverity.Warning:
		Events.RaiseEvent(E_TestComponent.WarningEvent);

	TcEventSeverity.Info:
		Events.RaiseEvent(E_TestComponent.InfoEvent);

	TcEventSeverity.Verbose:
		Events.RaiseEvent(E_TestComponent.VerboseEvent);
END_CASE
END_METHOD

METHOD Reset
Events.Reset();
END_METHOD

METHOD SetEventReactions
VAR_INPUT
	Verbose	 : DINT := 0;
	Info	 : DINT := 1;
	Warning	 : DINT := 2;
	Error	 : DINT := 3;
	Critical : DINT := 4;
END_VAR
Events.SetEventReactions(Verbose,
						 Info,
						 Warning,
						 Error,
						 Critical);
END_METHOD

END_FUNCTION_BLOCK

// ---- UnitTests/Statemachine/Statemachine_TEST.TcPOU
FUNCTION_BLOCK Statemachine_TEST
VAR
	Statemachine : Statemachine<1>('Test Statemachine');
	IdleState	 : State_Mockup(0, Statemachine);
	ExecuteState : State_Mockup(1, Statemachine);

	//
	TestState	  : State_Mockup(0, 0);
	StateList	  : StateList<ApplicationBaseParameter.MaxCountInCollections>;
	TestState2	  : State_Mockup(0, 0);
	Statemachine2 : Statemachine<1>('Test Statemachine');
END_VAR

ListAddGetState();
StatemachineVisitor();
StatemachineCollectionAccess();
CurrentState();
ChangeState();
StateExecuting();

METHOD ChangeState
VAR_INST
	Expected : DINT;
	Actual	 : DINT;
END_VAR
IF TestSuite.Test(__POUNAME()).ExecuteTest() THEN
	Expected := 1;
	Statemachine.States.AddStateAtIndex(0, IdleState);
	Statemachine.States.AddStateAtIndex(1, ExecuteState);
	Statemachine.CyclicLogic();
	Statemachine.ChangeState(1);
	Actual := Statemachine.CurrentState;
	TestSuite.Test(__POUNAME()).AssertEqual(Expected, Actual);
END_IF
END_METHOD

METHOD CurrentState
VAR_INST
	Expected : DINT;
	Actual	 : DINT;
END_VAR
IF TestSuite.Test(__POUNAME()).ExecuteTest() THEN
	Expected := 1;
	Statemachine.CyclicLogic();
	Actual := Statemachine.CurrentState;
	TestSuite.Test(__POUNAME()).AssertEqual(Expected, Actual);
END_IF
END_METHOD

METHOD ListAddGetState
VAR_INST
	Expected   : BOOL;
	Actual	   : BOOL;
	InputState : I_State;
	GetState   : I_State;
END_VAR
IF TestSuite.Test(__POUNAME()).ExecuteTest() THEN
	Expected   := TRUE;
	InputState := TestState;
	StateList.AddStateAtIndex(0, TestState);
	GetState := StateList.GetStateAtIndex(0);
	Actual	 := GetState = InputState;
	TestSuite.Test(__POUNAME()).AssertEqual(Expected, Actual);
END_IF
END_METHOD

METHOD StateExecuting
VAR_INST
	Expected : BOOL;
	Actual	 : BOOL;
END_VAR
IF TestSuite.Test(__POUNAME()).ExecuteTest() THEN
	Expected := TRUE;
	Statemachine.CyclicLogic();
	Actual := ExecuteState.IsExecuting;
	TestSuite.Test(__POUNAME()).AssertEqual(Expected, Actual);
END_IF
END_METHOD

METHOD StatemachineCollectionAccess
VAR_INST
	Expected   : BOOL;
	Actual	   : BOOL;
	InputState : I_State;
	GetState   : I_State;
END_VAR
IF TestSuite.Test(__POUNAME()).ExecuteTest() THEN
	Expected   := TRUE;
	InputState := TestState2;
	Statemachine2.States.AddStateAtIndex(1, TestState2);
	GetState := Statemachine2.States.GetStateAtIndex(1);
	Actual	 := GetState = InputState;
	TestSuite.Test(__POUNAME()).AssertEqual(Expected, Actual);
END_IF
END_METHOD

METHOD StatemachineVisitor
VAR_INST
	Expected			: STRING;
	Actual				: STRING;
	StateVisitor_Mockup : StateMachineVisitor_Mockup;
END_VAR
IF TestSuite.Test(__POUNAME()).ExecuteTest() THEN
	Expected := 'Test Statemachine';
	Statemachine.Accept(StateVisitor_Mockup);
	Actual := StateVisitor_Mockup.StatemachineName;
	TestSuite.Test(__POUNAME()).AssertEqual(Expected, Actual);
END_IF
END_METHOD

END_FUNCTION_BLOCK

// ---- _Mockups/Statemachine/State_Mockup.TcPOU
FUNCTION_BLOCK State_Mockup EXTENDS State
VAR
	_IsExecuting : BOOL;
END_VAR

METHOD Executing : BOOL
_IsExecuting := TRUE;
END_METHOD

PROPERTY IsExecuting : BOOL
GET
IsExecuting := _IsExecuting;
END_GET
END_PROPERTY

END_FUNCTION_BLOCK

// ---- _Mockups/Statemachine/StateMachineVisitor_Mockup.TcPOU
FUNCTION_BLOCK StateMachineVisitor_Mockup IMPLEMENTS I_ComponentVisitor
VAR
	_StatemachineName : T_MaxString;
END_VAR

PROPERTY StatemachineName : T_MaxString
GET
StatemachineName := _StatemachineName;
END_GET
END_PROPERTY

METHOD VisitComponent
VAR_INPUT
	Component : I_Component;
END_VAR

VAR
	Statemachine : I_Statemachine;
END_VAR
IF __QUERYINTERFACE(Component, Statemachine) THEN
	_StatemachineName := Statemachine.Name;
END_IF
END_METHOD

END_FUNCTION_BLOCK

// ---- UnitTests/Collection/Collection_TEST.TcPOU
FUNCTION_BLOCK Collection_TEST
VAR
	Collection : Collection_Mockup<3>;
	Item1	   : Item_Mockup;
	Item2	   : Item_Mockup;
	Item3	   : Item_Mockup;
END_VAR

AddTwoItems();
GetFirstItemById();
GetSecondItemById();
RemoveLastItem();
RemoveFirstItem();
RemoveToEmpty();
CheckCurrentIndexNull();
EnumeratorMoveNextFirst();
CheckCurrentIndex1();
EnumeratorMoveNextSecond();
CheckCurrentIndex2();
EnumeratorMoveNextThird();
CheckCurrentIndex3();
EnumeratorMoveNextEmpty();
EnumeratorReset();
Clear();

METHOD AddTwoItems
VAR_INST
	Expected : UDINT;
	Actual	 : UDINT;
END_VAR
IF TestSuite.Test(__POUNAME()).ExecuteTest() THEN
	Expected := 2;
	Collection.AddItem(Item1);
	Collection.AddItem(Item2);
	Actual := Collection.Count;
	Collection.AddItem(Item3);
	TestSuite.Test(__POUNAME()).AssertEqual(Expected, Actual);
END_IF
END_METHOD

METHOD CheckCurrentIndex1
VAR
	Expected : UDINT;
	Actual	 : UDINT;
END_VAR
IF TestSuite.Test(__POUNAME()).ExecuteTest() THEN
	Expected := 1;
	Actual	 := Collection.CurrentItem;
	TestSuite.Test(__POUNAME()).AssertEqual(Expected, Actual);
END_IF
END_METHOD

METHOD CheckCurrentIndex2
VAR
	Expected : UDINT;
	Actual	 : UDINT;
END_VAR
IF TestSuite.Test(__POUNAME()).ExecuteTest() THEN
	Expected := 2;
	Actual	 := Collection.CurrentItem;
	TestSuite.Test(__POUNAME()).AssertEqual(Expected, Actual);
END_IF
END_METHOD

METHOD CheckCurrentIndex3
VAR
	Expected : UDINT;
	Actual	 : UDINT;
END_VAR
IF TestSuite.Test(__POUNAME()).ExecuteTest() THEN
	Expected := 3;
	Actual	 := Collection.CurrentItem;
	TestSuite.Test(__POUNAME()).AssertEqual(Expected, Actual);
END_IF
END_METHOD

METHOD CheckCurrentIndexNull
VAR
	Expected : UDINT;
	Actual	 : UDINT;
END_VAR
IF TestSuite.Test(__POUNAME()).ExecuteTest() THEN
	Expected := 0;
	Actual	 := Collection.CurrentItem;
	TestSuite.Test(__POUNAME()).AssertEqual(Expected, Actual);
END_IF
END_METHOD

METHOD Clear
VAR
	Expected : UDINT;
	Actual	 : UDINT;
END_VAR
IF TestSuite.Test(__POUNAME()).ExecuteTest() THEN
	Expected := 0;
	Collection.Clear();
	Actual := Collection.Count;
	TestSuite.Test(__POUNAME()).AssertEqual(Expected, Actual);
END_IF
END_METHOD

METHOD EnumeratorMoveNextEmpty
VAR
	Expected   : BOOL;
	Actual	   : BOOL;
	Response   : BOOL;
	TargetItem : I_Base;
	ActualItem : I_Base;
END_VAR
IF TestSuite.Test(__POUNAME()).ExecuteTest() THEN
	Expected   := TRUE;
	TargetItem := Item3;
	Response   := Collection.MoveToNext;
	ActualItem := Collection.Current;
	Actual	   := (ActualItem = TargetItem) AND NOT Response;
	TestSuite.Test(__POUNAME()).AssertEqual(Expected, Actual);
END_IF
END_METHOD

METHOD EnumeratorMoveNextFirst
VAR
	Expected   : BOOL;
	Actual	   : BOOL;
	Response   : BOOL;
	TargetItem : I_Base;
	ActualItem : I_Base;
END_VAR
IF TestSuite.Test(__POUNAME()).ExecuteTest() THEN
	Expected   := TRUE;
	TargetItem := Item1;
	Collection.AddItem(Item1);
	Collection.AddItem(Item2);
	Collection.AddItem(Item3);
	Response   := Collection.MoveToNext;
	ActualItem := Collection.Current;
	Actual	   := (ActualItem = TargetItem) AND Response;
	TestSuite.Test(__POUNAME()).AssertEqual(Expected, Actual);
END_IF
END_METHOD

METHOD EnumeratorMoveNextSecond
VAR
	Expected   : BOOL;
	Actual	   : BOOL;
	Response   : BOOL;
	TargetItem : I_Base;
	ActualItem : I_Base;
END_VAR
IF TestSuite.Test(__POUNAME()).ExecuteTest() THEN
	Expected   := TRUE;
	TargetItem := Item2;
	Response   := Collection.MoveToNext;
	ActualItem := Collection.Current;
	Actual	   := (ActualItem = TargetItem) AND Response;
	TestSuite.Test(__POUNAME()).AssertEqual(Expected, Actual);
END_IF
END_METHOD

METHOD EnumeratorMoveNextThird
VAR
	Expected   : BOOL;
	Actual	   : BOOL;
	Response   : BOOL;
	TargetItem : I_Base;
	ActualItem : I_Base;
END_VAR
IF TestSuite.Test(__POUNAME()).ExecuteTest() THEN
	Expected   := TRUE;
	TargetItem := Item3;
	Response   := Collection.MoveToNext;
	ActualItem := Collection.Current;
	Actual	   := (ActualItem = TargetItem) AND Response;
	TestSuite.Test(__POUNAME()).AssertEqual(Expected, Actual);
END_IF
END_METHOD

METHOD EnumeratorReset
VAR
	Expected   : BOOL;
	Actual	   : BOOL;
	Response   : BOOL;
	TargetItem : I_Base;
	ActualItem : I_Base;
END_VAR
IF TestSuite.Test(__POUNAME()).ExecuteTest() THEN
	Expected   := TRUE;
	TargetItem := Item1;
	Collection.ResetIterator();
	Response   := Collection.MoveToNext;
	ActualItem := Collection.Current;
	Actual	   := (ActualItem = TargetItem) AND Response;
	TestSuite.Test(__POUNAME()).AssertEqual(Expected, Actual);
END_IF
END_METHOD

METHOD GetFirstItemById
VAR_INST
	Expected   : BOOL;
	Actual	   : BOOL;
	TargetItem : I_Base;
	ActualItem : I_Base;
END_VAR
IF TestSuite.Test(__POUNAME()).ExecuteTest() THEN
	Expected   := TRUE;
	TargetItem := Item1;
	ActualItem := Collection.GetItemByIndex(0);
	Actual	   := (TargetItem = ActualItem);
	TestSuite.Test(__POUNAME()).AssertEqual(Expected, Actual);
END_IF
END_METHOD

METHOD GetSecondItemById
VAR_INST
	Expected   : BOOL;
	Actual	   : BOOL;
	TargetItem : I_Base;
	ActualItem : I_Base;
END_VAR
IF TestSuite.Test(__POUNAME()).ExecuteTest() THEN
	Expected   := TRUE;
	TargetItem := Item2;
	ActualItem := Collection.GetItemByIndex(1);
	Actual	   := (TargetItem = ActualItem);
	TestSuite.Test(__POUNAME()).AssertEqual(Expected, Actual);
END_IF
END_METHOD

METHOD RemoveFirstItem
VAR_INST
	Expected   : BOOL;
	Actual	   : BOOL;
	TargetItem : I_Base;
	ActualItem : I_Base;
END_VAR
IF TestSuite.Test(__POUNAME()).ExecuteTest() THEN
	Expected   := TRUE;
	TargetItem := Item2;
	Collection.RemoveItem(Item1);
	ActualItem := Collection.GetItemByIndex(0);
	Actual	   := (TargetItem = ActualItem) AND (Collection.Count = 1);
	TestSuite.Test(__POUNAME()).AssertEqual(Expected, Actual);
END_IF
END_METHOD

METHOD RemoveLastItem
VAR_INST
	Expected   : BOOL;
	Actual	   : BOOL;
	TargetItem : I_Base;
	ActualItem : I_Base;
END_VAR
IF TestSuite.Test(__POUNAME()).ExecuteTest() THEN
	Expected   := TRUE;
	TargetItem := 0;
	Collection.RemoveItem(Item3);
	ActualItem := Collection.GetItemByIndex(2);
	Actual	   := (TargetItem = ActualItem) AND (Collection.Count = 2);
	TestSuite.Test(__POUNAME()).AssertEqual(Expected, Actual);
END_IF
END_METHOD

METHOD RemoveToEmpty
VAR_INST
	Expected : UDINT;
	Actual	 : UDINT;
END_VAR
IF TestSuite.Test(__POUNAME()).ExecuteTest() THEN
	Expected := 0;
	Collection.RemoveItem(Item2);
	Actual := Collection.Count;
	TestSuite.Test(__POUNAME()).AssertEqual(Expected, Actual);
END_IF
END_METHOD

END_FUNCTION_BLOCK

// ---- _Mockups/Collection/Collection_Mockup.TcPOU
FUNCTION_BLOCK Collection_Mockup
VAR_GENERIC CONSTANT
	MockupSize : UDINT := 2;
END_VAR
EXTENDS Collection<MockupSize>
VAR
END_VAR

METHOD GetItemByIndex : I_Base
VAR_INPUT
	Index : UDINT;
END_VAR
GetItemByIndex := _Data[Index];
END_METHOD

END_FUNCTION_BLOCK

// ---- _Mockups/Collection/Item_Mockup.TcPOU
FUNCTION_BLOCK Item_Mockup IMPLEMENTS I_Base
VAR
	_Name : T_MaxString;
END_VAR

PROPERTY Name : T_MaxString
GET
Name := _Name;
END_GET
SET
_Name := Name;
END_SET
END_PROPERTY

END_FUNCTION_BLOCK

// ---- UnitTests/List/List_TEST.TcPOU
FUNCTION_BLOCK List_TEST
VAR
	List  : List<5>;
	Item1 : Item_Mockup;
	Item2 : Item_Mockup;
	Item3 : Item_Mockup;
END_VAR

InsertByIndex();
InsertByIndexFail();
InsertByIndexShift();
GetByIndex();
ContainsItemTrue();
ContainsItemFalse();
RemoveItemByIndex();
Clear();
AddTwoItems();
RemoveFirstItem();
RemoveLastItem();
RemoveToEmpty();
ContainsAfterItemRemoval();
RemoveDuplicateItems();
ContainsOnEmptyList();
Test();
InsertIndex0Shift();

METHOD AddTwoItems
VAR_INST
	Expected : UDINT;
	Actual	 : UDINT;
END_VAR
IF TestSuite.Test(__POUNAME()).ExecuteTest() THEN
	Expected := 2;
	List.Clear();
	List.AddItem(Item1);
	List.AddItem(Item2);
	Actual := List.Count;
	List.AddItem(Item3);
	TestSuite.Test(__POUNAME()).AssertEqual(Expected, Actual);
END_IF
END_METHOD

METHOD Clear
VAR
	Expected : UDINT;
	Actual	 : UDINT;
END_VAR
IF TestSuite.Test(__POUNAME()).ExecuteTest() THEN
	Expected := 0;
	List.Clear();
	Actual := List.Count;
	TestSuite.Test(__POUNAME()).AssertEqual(Expected, Actual);
END_IF
END_METHOD

METHOD ContainsAfterItemRemoval
VAR
	Expected	 : BOOL;
	Actual		 : BOOL;
	ExpectedItem : I_Base;
	ActualItem	 : I_Base;
END_VAR
IF TestSuite.Test(__POUNAME()).ExecuteTest() THEN
	Expected	 := TRUE;
	ExpectedItem := Item2;
	List.Clear();
	ExpectedItem := Item2;
	List.AddItem(Item1);
	List.AddItem(Item2);
	List.RemoveItem(Item1);
	ActualItem := List.GetAtIndex(0);
	Actual	   := ExpectedItem = ActualItem;
	TestSuite.Test(__POUNAME()).AssertEqual(Expected, Actual);

	//cleanup
	List.Clear();
END_IF
END_METHOD

METHOD ContainsItemFalse
VAR
	Expected : BOOL;
	Actual	 : BOOL;
END_VAR
IF TestSuite.Test(__POUNAME()).ExecuteTest() THEN
	Expected := FALSE;
	Actual	 := List.ContainsItem(Item3);
	TestSuite.Test(__POUNAME()).AssertEqual(Expected, Actual);
END_IF
END_METHOD

METHOD ContainsItemTrue
VAR
	Expected : BOOL;
	Actual	 : BOOL;
END_VAR
IF TestSuite.Test(__POUNAME()).ExecuteTest() THEN
	Expected := TRUE;
	Actual	 := List.ContainsItem(Item2);
	TestSuite.Test(__POUNAME()).AssertEqual(Expected, Actual);
END_IF
END_METHOD

METHOD ContainsOnEmptyList
VAR
	Expected : BOOL;
	Actual	 : BOOL;
END_VAR
IF TestSuite.Test(__POUNAME()).ExecuteTest() THEN
	Expected := FALSE;
	List.Clear();
	Actual := List.ContainsItem(Item1);
	TestSuite.Test(__POUNAME()).AssertEqual(Expected, Actual);
END_IF
END_METHOD

METHOD GetByIndex
VAR
	Expected   : BOOL;
	Actual	   : BOOL;
	TargetItem : I_Base;
	ActualItem : I_Base;
END_VAR
IF TestSuite.Test(__POUNAME()).ExecuteTest() THEN
	Expected   := TRUE;
	TargetItem := Item2;
	ActualItem := List.GetAtIndex(1);
	Actual	   := TargetItem = ActualItem;
	TestSuite.Test(__POUNAME()).AssertEqual(Expected, Actual);
END_IF
END_METHOD

METHOD InsertByIndex
VAR
	Expected   : UDINT;
	Actual	   : UDINT;
	TargetItem : I_Base;
	ActualItem : I_Base;
END_VAR
IF TestSuite.Test(__POUNAME()).ExecuteTest() THEN
	Expected := 1;
	List.InsertAtIndex(Item2, 0);
	Actual := List.Count;
	TestSuite.Test(__POUNAME()).AssertEqual(Expected, Actual);
END_IF
END_METHOD

METHOD InsertByIndexFail
VAR
	Expected : BOOL;
	Actual	 : BOOL;
END_VAR
IF TestSuite.Test(__POUNAME()).ExecuteTest() THEN
	Expected := FALSE;
	Actual	 := List.InsertAtIndex(Item2, 2);
	TestSuite.Test(__POUNAME()).AssertEqual(Expected, Actual);
END_IF
END_METHOD

METHOD InsertByIndexShift
VAR
	Expected   : UDINT;
	Actual	   : UDINT;
	TargetItem : I_Base;
	ActualItem : I_Base;
END_VAR
IF TestSuite.Test(__POUNAME()).ExecuteTest() THEN
	Expected := 2;
	List.InsertAtIndex(Item1, 0);
	Actual := List.Count;
	TestSuite.Test(__POUNAME()).AssertEqual(Expected, Actual);
END_IF
END_METHOD

METHOD InsertIndex0Shift
VAR
	Expected	  : BOOL;
	Actual		  : BOOL;
	ExpectedItems : ARRAY[0..4] OF I_Base;
	ActualItems	  : ARRAY[0..4] OF I_Base;
	Item4		  : Item_Mockup;
	Item5		  : Item_Mockup;
	i			  : UDINT;
END_VAR
IF TestSuite.Test(__POUNAME()).ExecuteTest() THEN
	Expected		 := TRUE;
	ExpectedItems[0] := Item5;
	ExpectedItems[1] := Item1;
	ExpectedItems[2] := Item2;
	ExpectedItems[3] := Item3;
	ExpectedItems[4] := Item4;
	List.Clear();
	FOR i := 1 TO 4 DO
		List.AddItem(ExpectedItems[i]);
	END_FOR

	List.InsertAtIndex(Item5, 0);
	Actual := TRUE;
	FOR i := 0 TO 4 DO
		ActualItems[i] := List.GetAtIndex(i);
		Actual		   := Actual AND ExpectedItems[i] = ActualItems[i];
	END_FOR

	TestSuite.Test(__POUNAME()).AssertEqual(Expected, Actual);

	//cleanup
	List.Clear();
END_IF
END_METHOD

METHOD RemoveDuplicateItems
VAR
	Expected   : UDINT;
	Actual	   : UDINT;
	TargetItem : I_Base;
	ActualItem : I_Base;
END_VAR
IF TestSuite.Test(__POUNAME()).ExecuteTest() THEN
	Expected   := 1;
	TargetItem := Item2;
	List.Clear();
	List.AddItem(Item1);
	List.AddItem(Item1);
	List.AddItem(Item2);
	List.RemoveItem(Item1);
	Actual := List.Count;
	TestSuite.Test(__POUNAME()).AssertEqual(Expected, Actual);

	//cleanup
	List.Clear();
END_IF
END_METHOD

METHOD RemoveFirstItem
VAR_INST
	Expected   : BOOL;
	Actual	   : BOOL;
	TargetItem : I_Base;
	ActualItem : I_Base;
END_VAR
IF TestSuite.Test(__POUNAME()).ExecuteTest() THEN
	Expected   := TRUE;
	TargetItem := Item2;
	List.RemoveItem(Item1);
	ActualItem := List.GetAtIndex(0);
	Actual	   := (TargetItem = ActualItem) AND (List.Count = 2);
	TestSuite.Test(__POUNAME()).AssertEqual(Expected, Actual);
END_IF
END_METHOD

METHOD RemoveItemByIndex
VAR
	Expected   : UDINT;
	Actual	   : UDINT;
	TargetItem : I_Base;
	ActualItem : I_Base;
END_VAR
IF TestSuite.Test(__POUNAME()).ExecuteTest() THEN
	Expected := 1;
	List.RemoveAtIndex(1);
	Actual := List.Count;
	TestSuite.Test(__POUNAME()).AssertEqual(Expected, Actual);
END_IF
END_METHOD

METHOD RemoveLastItem
VAR_INST
	Expected   : BOOL;
	Actual	   : BOOL;
	TargetItem : I_Base;
	ActualItem : I_Base;
END_VAR
IF TestSuite.Test(__POUNAME()).ExecuteTest() THEN
	Expected   := TRUE;
	TargetItem := 0;
	List.RemoveItem(Item3);
	ActualItem := List.GetAtIndex(2);
	Actual	   := (TargetItem = ActualItem) AND (List.Count = 1);
	TestSuite.Test(__POUNAME()).AssertEqual(Expected, Actual);
END_IF
END_METHOD

METHOD RemoveToEmpty
VAR_INST
	Expected : UDINT;
	Actual	 : UDINT;
END_VAR
IF TestSuite.Test(__POUNAME()).ExecuteTest() THEN
	Expected := 0;
	List.RemoveItem(Item2);
	Actual := List.Count;
	TestSuite.Test(__POUNAME()).AssertEqual(Expected, Actual);
END_IF
END_METHOD

METHOD Test
VAR
	Expected	 : BOOL;
	Actual		 : BOOL;
	ExpectedItem : I_Base;
	ActualItem	 : I_Base;
END_VAR
IF TestSuite.Test(__POUNAME()).ExecuteTest() THEN
	Expected	 := TRUE;
	ExpectedItem := Item2;
	List.Clear();
	List.AddItem(Item1);
	List.AddItem(Item2);
	List.RemoveAtIndex(0);
	ActualItem := List.GetAtIndex(0);
	Actual	   := ActualItem = ExpectedItem;
	TestSuite.Test(__POUNAME()).AssertEqual(Expected, Actual);

	//cleanup
	List.Clear();
END_IF
END_METHOD

END_FUNCTION_BLOCK

// ---- UnitTests/ModeChange/ModeControl_TEST.TcPOU
FUNCTION_BLOCK ModeControl_TEST
VAR
END_VAR

// Call test methods
DefaultMode();
ChangeValidMode();
ChangeInvalidMode();
MultipleModesChange();

METHOD ChangeInvalidMode
VAR_INST
	Expected : DINT;
	Actual	 : DINT;
	TestMode : DINT;
END_VAR
VAR
	ModeControl : ModeControl_Mockup;
END_VAR
IF TestSuite.Test(__POUNAME()).ExecuteTest() THEN
	IF ModeControl._CurrentMode = 1 THEN
		TestMode := 0;
		ModeControl.ChangeMode(TestMode);
		Expected := 1; // Should remain at default
		Actual	 := ModeControl._CurrentMode;
		TestSuite.Test(__POUNAME()).AssertEqual(Expected, Actual);
	ELSE
		ModeControl.ChangeMode(1);
	END_IF
END_IF
END_METHOD

METHOD ChangeValidMode
VAR_INST
	Expected : DINT;
	Actual	 : DINT;
	TestMode : DINT;
END_VAR
VAR
	ModeControl : ModeControl_Mockup;
END_VAR
IF TestSuite.Test(__POUNAME()).ExecuteTest() THEN
	TestMode := 5;
	ModeControl.ChangeMode(TestMode);
	Expected := TestMode;
	Actual	 := ModeControl._CurrentMode;
	TestSuite.Test(__POUNAME()).AssertEqual(Expected, Actual);
END_IF
END_METHOD

METHOD DefaultMode
VAR_INST
	Expected : DINT;
	Actual	 : DINT;
END_VAR
VAR
	ModeControl : ModeControl_Mockup;
END_VAR
IF TestSuite.Test(__POUNAME()).ExecuteTest() THEN
	Expected := 1;
	Actual	 := ModeControl._CurrentMode;
	TestSuite.Test(__POUNAME()).AssertEqual(Expected, Actual);
END_IF
END_METHOD

METHOD MultipleModesChange
VAR_INST
	Expected : DINT;
	Actual	 : DINT;
	TestMode : DINT;
END_VAR
VAR
	ModeControl : ModeControl_Mockup;
END_VAR
IF TestSuite.Test(__POUNAME()).ExecuteTest() THEN
	TestMode := 3;
	ModeControl.ChangeMode(TestMode);
	TestMode := 7;
	ModeControl.ChangeMode(TestMode);
	Expected := TestMode;
	Actual	 := ModeControl._CurrentMode;
	TestSuite.Test(__POUNAME()).AssertEqual(Expected, Actual);
END_IF
END_METHOD

END_FUNCTION_BLOCK

// ---- _Mockups/ModeChange/ModeControl_Mockup.TcPOU
FUNCTION_BLOCK ModeControl_Mockup EXTENDS ModeControl
VAR
	{attribute 'hide'}
	_IsChangeModeInvoked : BOOL;
	{attribute 'hide'}
	_LastRequestedMode : DINT;
	{attribute 'hide'}
	_IsExecuting : BOOL;
END_VAR

// Override the ChangeMode method to add mockup tracking
METHOD ChangeMode
VAR_INPUT
	RequestedMode : DINT;
END_VAR
_IsChangeModeInvoked := TRUE;
_LastRequestedMode	 := RequestedMode;
_IsExecuting		 := TRUE;

// Call the base implementation
SUPER^.ChangeMode(RequestedMode);
END_METHOD

// Method to complete/reset execution state
METHOD Complete
_IsExecuting		 := FALSE;
_IsChangeModeInvoked := FALSE;
_LastRequestedMode	 := 0;
END_METHOD

// Mockup specific method to simulate execution state
METHOD Executing
_IsExecuting := TRUE;
END_METHOD

// Additional method to check if ChangeMode was called
METHOD IsExecuting : BOOL
IsExecuting := _IsExecuting;
END_METHOD

END_FUNCTION_BLOCK

// ---- UnitTests/CollectionPeeker/CollectionPeeker_Test.TcPOU
FUNCTION_BLOCK CollectionPeeker_Test
VAR
	ComponentArray : ARRAY[0..9] OF Component_Mockup[(Name := '1'), (Name := '2'), (Name := '3'), (Name := '4'), (Name := '5'), (Name := '6'), (Name := '7'), (Name := '8'), (Name := '9'), (Name := '10')];
	AllComponents  : Collection<20>;
	i			   : UDINT;
END_VAR

IF AllComponents.Count <> (SIZEOF(ComponentArray) / SIZEOF(ComponentArray[0])) THEN
	FOR i := 0 TO (SIZEOF(ComponentArray) / SIZEOF(ComponentArray[0])) - 1 DO
		AllComponents.AddItem(ComponentArray[i]);
	END_FOR
END_IF

SetCollectionCheck();
SetFirstItem();
MoveDownOne();
MoveUpOne();
PageDownOne();
PageUpOne();
MoveUpOneRollOver();
MoveDownOneRollOver();
PageUpRollOver();
PageDownRollOver();
NoCollection();
CollectionSmallerThanPeekSize();

METHOD CollectionSmallerThanPeekSize
VAR
	Expected		 : BOOL;
	Actual			 : BOOL;
	NamesEqual		 : BOOL;
	ExpectedNames	 : ARRAY[1..10] OF STRING[5];
	ActualNames		 : ARRAY[1..10] OF STRING[5];
	CurrentComponent : I_Component;

	//
	Peeker		   : CollectionPeeker_Mock<12>;
	CollectionName : T_MaxString;
	i			   : UDINT;
END_VAR
IF TestSuite.Test(__POUNAME()).ExecuteTest() THEN
	Expected			  := TRUE;
	CollectionName		  := 'Test Collection';
	ExpectedNames[1]	  := ComponentArray[0].Name;
	ExpectedNames[2]	  := ComponentArray[1].Name;
	ExpectedNames[3]	  := ComponentArray[2].Name;
	ExpectedNames[4]	  := ComponentArray[3].Name;
	ExpectedNames[5]	  := ComponentArray[4].Name;
	ExpectedNames[6]	  := ComponentArray[5].Name;
	ExpectedNames[7]	  := ComponentArray[6].Name;
	ExpectedNames[8]	  := ComponentArray[7].Name;
	ExpectedNames[9]	  := ComponentArray[8].Name;
	ExpectedNames[10]	  := ComponentArray[9].Name;
	Peeker.CollectionName := CollectionName;
	Peeker.PeekCollection(AllComponents);
	Peeker.MoveDownOne := TRUE;
	Peeker.MoveDownOne := TRUE;
	Peeker.MoveUpOne   := TRUE;
	Peeker.PageDown	   := TRUE;
	Peeker.PageUp	   := TRUE;
	NamesEqual		   := TRUE;
	FOR i := 1 TO 10 DO
		__QUERYINTERFACE(Peeker.Items[i], CurrentComponent);
		ActualNames[i] := CurrentComponent.Name;
		NamesEqual	   := NamesEqual AND ActualNames[i] = ExpectedNames[i];
	END_FOR

	Actual := Peeker.FirstItem = 1 AND Peeker.LastItem = 12 AND NamesEqual;
	TestSuite.Test(__POUNAME()).AssertEqual(Expected, Actual);
END_IF
END_METHOD

METHOD MoveDownOne
VAR
	Expected		 : BOOL;
	Actual			 : BOOL;
	NamesEqual		 : BOOL;
	ExpectedNames	 : ARRAY[1..5] OF STRING[5];
	ActualNames		 : ARRAY[1..5] OF STRING[5];
	CurrentComponent : I_Component;

	//
	Peeker		   : CollectionPeeker_Mock<5>;
	CollectionName : T_MaxString;
	i			   : UDINT;
END_VAR
IF TestSuite.Test(__POUNAME()).ExecuteTest() THEN
	Expected			  := TRUE;
	CollectionName		  := 'Test Collection';
	ExpectedNames[1]	  := ComponentArray[1].Name;
	ExpectedNames[2]	  := ComponentArray[2].Name;
	ExpectedNames[3]	  := ComponentArray[3].Name;
	ExpectedNames[4]	  := ComponentArray[4].Name;
	ExpectedNames[5]	  := ComponentArray[5].Name;
	Peeker.CollectionName := CollectionName;
	Peeker.PeekCollection(AllComponents);
	Peeker.MoveDownOne := TRUE;
	NamesEqual		   := TRUE;
	FOR i := 1 TO 5 DO
		__QUERYINTERFACE(Peeker.Items[i], CurrentComponent);
		ActualNames[i] := CurrentComponent.Name;
		NamesEqual	   := NamesEqual AND ActualNames[i] = ExpectedNames[i];
	END_FOR

	Actual := Peeker.FirstItem = 2 AND Peeker.LastItem = 6 AND NamesEqual;
	TestSuite.Test(__POUNAME()).AssertEqual(Expected, Actual);
END_IF
END_METHOD

METHOD MoveDownOneRollOver
VAR
	Expected		 : BOOL;
	Actual			 : BOOL;
	NamesEqual		 : BOOL;
	ExpectedNames	 : ARRAY[1..5] OF STRING[5];
	ActualNames		 : ARRAY[1..5] OF STRING[5];
	CurrentComponent : I_Component;

	//
	Peeker		   : CollectionPeeker_Mock<5>;
	CollectionName : T_MaxString;
	i			   : UDINT;
END_VAR
IF TestSuite.Test(__POUNAME()).ExecuteTest() THEN
	Expected			  := TRUE;
	CollectionName		  := 'Test Collection';
	ExpectedNames[1]	  := ComponentArray[6].Name;
	ExpectedNames[2]	  := ComponentArray[7].Name;
	ExpectedNames[3]	  := ComponentArray[8].Name;
	ExpectedNames[4]	  := ComponentArray[9].Name;
	ExpectedNames[5]	  := ComponentArray[0].Name;
	Peeker.CollectionName := CollectionName;
	Peeker.PeekCollection(AllComponents);
	Peeker.FirstItem   := 6;
	Peeker.MoveDownOne := TRUE;
	NamesEqual		   := TRUE;
	FOR i := 1 TO 5 DO
		__QUERYINTERFACE(Peeker.Items[i], CurrentComponent);
		ActualNames[i] := CurrentComponent.Name;
		NamesEqual	   := NamesEqual AND ActualNames[i] = ExpectedNames[i];
	END_FOR

	Actual := Peeker.FirstItem = 7 AND Peeker.LastItem = 1 AND NamesEqual;
	TestSuite.Test(__POUNAME()).AssertEqual(Expected, Actual);
END_IF
END_METHOD

METHOD MoveUpOne
VAR
	Expected		 : BOOL;
	Actual			 : BOOL;
	NamesEqual		 : BOOL;
	ExpectedNames	 : ARRAY[1..5] OF STRING[5];
	ActualNames		 : ARRAY[1..5] OF STRING[5];
	CurrentComponent : I_Component;

	//
	Peeker		   : CollectionPeeker_Mock<5>;
	CollectionName : T_MaxString;
	i			   : UDINT;
END_VAR
IF TestSuite.Test(__POUNAME()).ExecuteTest() THEN
	Expected			  := TRUE;
	CollectionName		  := 'Test Collection';
	ExpectedNames[1]	  := ComponentArray[1].Name;
	ExpectedNames[2]	  := ComponentArray[2].Name;
	ExpectedNames[3]	  := ComponentArray[3].Name;
	ExpectedNames[4]	  := ComponentArray[4].Name;
	ExpectedNames[5]	  := ComponentArray[5].Name;
	Peeker.CollectionName := CollectionName;
	Peeker.PeekCollection(AllComponents);
	Peeker.FirstItem := 3;
	Peeker.MoveUpOne := TRUE;
	NamesEqual		 := TRUE;
	FOR i := 1 TO 5 DO
		__QUERYINTERFACE(Peeker.Items[i], CurrentComponent);
		ActualNames[i] := CurrentComponent.Name;
		NamesEqual	   := NamesEqual AND ActualNames[i] = ExpectedNames[i];
	END_FOR

	Actual := Peeker.FirstItem = 2 AND Peeker.LastItem = 6 AND NamesEqual;
	TestSuite.Test(__POUNAME()).AssertEqual(Expected, Actual);
END_IF
END_METHOD

METHOD MoveUpOneRollOver
VAR
	Expected		 : BOOL;
	Actual			 : BOOL;
	NamesEqual		 : BOOL;
	ExpectedNames	 : ARRAY[1..5] OF STRING[5];
	ActualNames		 : ARRAY[1..5] OF STRING[5];
	CurrentComponent : I_Component;

